LIN {X 0,Y 552.339,Z 586.998,A -85,B 0,C 180,E1 25712.762,E2 25712.762} C_VEL
LIN {X 0,Y 551.347,Z 587.125,A -85,B 0,C 180,E1 25711.964,E2 25711.964} C_VEL
LIN {X 0,Y 544.942,Z 587.913,A -85,B 0,C 180,E1 25709.72,E2 25709.72} C_VEL
LIN {X 0,Y 544.404,Z 587.984,A -85,B 0,C 180,E1 25709.136,E2 25709.136} C_VEL
LIN {X 0,Y 544.37,Z 587.986,A -85,B 0,C 180,E1 25705.803,E2 25705.803} C_VEL
LIN {X 0,Y 544.404,Z 587.987,A -85,B 0,C 180,E1 25702.428,E2 25702.428} C_VEL
LIN {X 0,Y 544.416,Z 588.083,A -85,B 0,C 180,E1 25698.94,E2 25698.94} C_VEL
LIN {X 0,Y 547.399,Z 600.07,A -85,B 0,C 180,E1 25697.246,E2 25697.246} C_VEL
LIN {X 0,Y 546.491,Z 629.146,A -85,B 0,C 180,E1 25693.756,E2 25693.756} C_VEL
LIN {X 0,Y 545.718,Z 658.309,A -85,B 0,C 180,E1 25690.342,E2 25690.342} C_VEL
LIN {X 0,Y 545.195,Z 688.021,A -85,B 0,C 180,E1 25686.98,E2 25686.98} C_VEL
LIN {X 0,Y 544.902,Z 710.009,A -85,B 0,C 180,E1 25684.567,E2 25684.567} C_VEL
LIN {X 0,Y 545.702,Z 718.325,A -85,B 0,C 180,E1 25684.417,E2 25684.417} C_VEL
LIN {X 0,Y 545.347,Z 821.497,A -85,B 0,C 180,E1 25683.028,E2 25683.028} C_VEL
LIN {X 0,Y 545.212,Z 836.514,A -85,B 0,C 180,E1 25682.627,E2 25682.627} C_VEL
LIN {X 0,Y 544.998,Z 851.155,A -85,B 0,C 180,E1 25682.019,E2 25682.019} C_VEL
LIN {X 0,Y 544.754,Z 864.801,A -85,B 0,C 180,E1 25681.232,E2 25681.232} C_VEL
LIN {X 0,Y 544.523,Z 876.818,A -85,B 0,C 180,E1 25680.329,E2 25680.329} C_VEL
LIN {X 0,Y 544.331,Z 888.046,A -85,B 0,C 180,E1 25679.248,E2 25679.248} C_VEL
LIN {X 0,Y 544.163,Z 897.795,A -85,B 0,C 180,E1 25678.059,E2 25678.059} C_VEL
LIN {X 0,Y 544.036,Z 906.382,A -85,B 0,C 180,E1 25676.721,E2 25676.721} C_VEL
LIN {X 0,Y 543.965,Z 913.553,A -85,B 0,C 180,E1 25675.242,E2 25675.242} C_VEL
LIN {X 0,Y 543.93,Z 918.751,A -85,B 0,C 180,E1 25673.732,E2 25673.732} C_VEL
LIN {X 0,Y 543.919,Z 922.084,A -85,B 0,C 180,E1 25672.252,E2 25672.252} C_VEL
LIN {X 0,Y 543.917,Z 923.807,A -85,B 0,C 180,E1 25670.662,E2 25670.662} C_VEL
LIN {X 0,Y 543.917,Z 923.713,A -85,B 0,C 180,E1 25669.099,E2 25669.099} C_VEL
LIN {X 0,Y 543.919,Z 921.897,A -85,B 0,C 180,E1 25667.546,E2 25667.546} C_VEL
LIN {X 0,Y 543.934,Z 917.94,A -85,B 0,C 180,E1 25665.896,E2 25665.896} C_VEL
LIN {X 0,Y 543.976,Z 912.247,A -85,B 0,C 180,E1 25664.367,E2 25664.367} C_VEL
LIN {X 0,Y 544.045,Z 905.689,A -85,B 0,C 180,E1 25663.065,E2 25663.065} C_VEL
LIN {X 0,Y 544.186,Z 896.405,A -85,B 0,C 180,E1 25661.66,E2 25661.66} C_VEL
LIN {X 0,Y 544.379,Z 885.783,A -85,B 0,C 180,E1 25660.423,E2 25660.423} C_VEL
LIN {X 0,Y 544.567,Z 874.019,A -85,B 0,C 180,E1 25659.351,E2 25659.351} C_VEL
LIN {X 0,Y 544.808,Z 862.012,A -85,B 0,C 180,E1 25658.496,E2 25658.496} C_VEL
LIN {X 0,Y 545.046,Z 848.15,A -85,B 0,C 180,E1 25657.749,E2 25657.749} C_VEL
LIN {X 0,Y 545.235,Z 834.039,A -85,B 0,C 180,E1 25657.204,E2 25657.204} C_VEL
LIN {X 0,Y 545.374,Z 818.941,A -85,B 0,C 180,E1 25656.832,E2 25656.832} C_VEL
LIN {X 0,Y 545.482,Z 714.402,A -85,B 0,C 180,E1 25655.434,E2 25655.434} C_VEL
LIN {X 0,Y 544.878,Z 709.572,A -85,B 0,C 180,E1 25655.317,E2 25655.317} C_VEL
LIN {X 0,Y 545.341,Z 678.781,A -85,B 0,C 180,E1 25651.891,E2 25651.891} C_VEL
LIN {X 0,Y 545.944,Z 649.394,A -85,B 0,C 180,E1 25648.531,E2 25648.531} C_VEL
LIN {X 0,Y 546.652,Z 620.644,A -85,B 0,C 180,E1 25645.173,E2 25645.173} C_VEL
LIN {X 0,Y 547.193,Z 598.729,A -85,B 0,C 180,E1 25642.545,E2 25642.545} C_VEL
LIN {X 0,Y 544.402,Z 588.081,A -85,B 0,C 180,E1 25641.018,E2 25641.018} C_VEL
LIN {X 0,Y 544.396,Z 587.986,A -85,B 0,C 180,E1 25637.591,E2 25637.591} C_VEL
LIN {X 0,Y 544.389,Z 587.981,A -85,B 0,C 180,E1 25634.117,E2 25634.117} C_VEL
LIN {X 0,Y 544.391,Z 587.983,A -85,B 0,C 180,E1 25630.743,E2 25630.743} C_VEL
LIN {X 0,Y 544.383,Z 587.984,A -85,B 0,C 180,E1 25627.426,E2 25627.426} C_VEL
LIN {X 0,Y 544.4,Z 587.979,A -85,B 0,C 180,E1 25623.962,E2 25623.962} C_VEL
LIN {X 0,Y 544.398,Z 587.974,A -85,B 0,C 180,E1 25620.513,E2 25620.513} C_VEL
LIN {X 0,Y 544.377,Z 587.976,A -85,B 0,C 180,E1 25617.191,E2 25617.191} C_VEL
LIN {X 0,Y 544.397,Z 587.98,A -85,B 0,C 180,E1 25613.874,E2 25613.874} C_VEL
LIN {X 0,Y 544.388,Z 587.986,A -85,B 0,C 180,E1 25610.48,E2 25610.48} C_VEL
LIN {X 0,Y 544.379,Z 587.976,A -85,B 0,C 180,E1 25606.971,E2 25606.971} C_VEL
LIN {X 0,Y 544.399,Z 587.983,A -85,B 0,C 180,E1 25603.644,E2 25603.644} C_VEL
LIN {X 0,Y 544.372,Z 587.978,A -85,B 0,C 180,E1 25600.281,E2 25600.281} C_VEL
LIN {X 0,Y 544.399,Z 587.979,A -85,B 0,C 180,E1 25596.912,E2 25596.912} C_VEL
LIN {X 0,Y 544.405,Z 587.979,A -85,B 0,C 180,E1 25593.435,E2 25593.435} C_VEL
LIN {X 0,Y 544.368,Z 587.984,A -85,B 0,C 180,E1 25590.095,E2 25590.095} C_VEL
LIN {X 0,Y 544.401,Z 587.972,A -85,B 0,C 180,E1 25586.797,E2 25586.797} C_VEL
LIN {X 0,Y 544.37,Z 587.983,A -85,B 0,C 180,E1 25583.489,E2 25583.489} C_VEL
LIN {X 0,Y 544.387,Z 587.978,A -85,B 0,C 180,E1 25580.088,E2 25580.088} C_VEL
LIN {X 0,Y 544.402,Z 587.979,A -85,B 0,C 180,E1 25576.759,E2 25576.759} C_VEL
LIN {X 0,Y 544.364,Z 587.983,A -85,B 0,C 180,E1 25573.49,E2 25573.49} C_VEL
LIN {X 0,Y 544.402,Z 587.973,A -85,B 0,C 180,E1 25570.155,E2 25570.155} C_VEL
LIN {X 0,Y 544.361,Z 587.982,A -85,B 0,C 180,E1 25566.857,E2 25566.857} C_VEL
LIN {X 0,Y 544.387,Z 587.979,A -85,B 0,C 180,E1 25563.475,E2 25563.475} C_VEL
LIN {X 0,Y 544.404,Z 587.978,A -85,B 0,C 180,E1 25560.105,E2 25560.105} C_VEL
LIN {X 0,Y 544.358,Z 587.984,A -85,B 0,C 180,E1 25556.841,E2 25556.841} C_VEL
LIN {X 0,Y 544.406,Z 587.973,A -85,B 0,C 180,E1 25553.521,E2 25553.521} C_VEL
LIN {X 0,Y 544.353,Z 587.985,A -85,B 0,C 180,E1 25550.271,E2 25550.271} C_VEL
LIN {X 0,Y 544.395,Z 587.977,A -85,B 0,C 180,E1 25546.944,E2 25546.944} C_VEL
LIN {X 0,Y 544.373,Z 587.985,A -85,B 0,C 180,E1 25543.679,E2 25543.679} C_VEL
LIN {X 0,Y 544.359,Z 587.981,A -85,B 0,C 180,E1 25540.247,E2 25540.247} C_VEL
LIN {X 0,Y 544.409,Z 587.984,A -85,B 0,C 180,E1 25536.947,E2 25536.947} C_VEL
LIN {X 0,Y 544.346,Z 587.982,A -85,B 0,C 180,E1 25533.685,E2 25533.685} C_VEL
LIN {X 0,Y 544.406,Z 587.979,A -85,B 0,C 180,E1 25530.393,E2 25530.393} C_VEL
LIN {X 0,Y 544.355,Z 587.988,A -85,B 0,C 180,E1 25527.191,E2 25527.191} C_VEL
LIN {X 0,Y 544.362,Z 587.984,A -85,B 0,C 180,E1 25523.74,E2 25523.74} C_VEL
LIN {X 0,Y 544.405,Z 587.986,A -85,B 0,C 180,E1 25520.478,E2 25520.478} C_VEL
LIN {X 0,Y 544.342,Z 587.987,A -85,B 0,C 180,E1 25517.186,E2 25517.186} C_VEL
LIN {X 0,Y 544.409,Z 587.983,A -85,B 0,C 180,E1 25513.95,E2 25513.95} C_VEL
LIN {X 0,Y 544.343,Z 587.988,A -85,B 0,C 180,E1 25510.698,E2 25510.698} C_VEL
LIN {X 0,Y 544.397,Z 587.982,A -85,B 0,C 180,E1 25507.44,E2 25507.44} C_VEL
LIN {X 0,Y 544.362,Z 587.993,A -85,B 0,C 180,E1 25504.198,E2 25504.198} C_VEL
LIN {X 0,Y 544.39,Z 588.207,A -85,B 0,C 180,E1 25502.928,E2 25502.928} C_VEL
LIN {X 0,Y 549.723,Z 603.754,A -85,B 0,C 180,E1 25501.345,E2 25501.345} C_VEL
LIN {X 0,Y 548.818,Z 646.737,A -85,B 0,C 180,E1 25498.214,E2 25498.214} C_VEL
LIN {X 0,Y 547.856,Z 691.846,A -85,B 0,C 180,E1 25494.939,E2 25494.939} C_VEL
LIN {X 0,Y 549.107,Z 701.947,A -85,B 0,C 180,E1 25494.729,E2 25494.729} C_VEL
LIN {X 0,Y 548.003,Z 901.303,A -85,B 0,C 180,E1 25491.965,E2 25491.965} C_VEL
LIN {X 0,Y 547.684,Z 920.34,A -85,B 0,C 180,E1 25491.503,E2 25491.503} C_VEL
LIN {X 0,Y 547.305,Z 938.39,A -85,B 0,C 180,E1 25490.87,E2 25490.87} C_VEL
LIN {X 0,Y 546.826,Z 956.036,A -85,B 0,C 180,E1 25490.05,E2 25490.05} C_VEL
LIN {X 0,Y 546.332,Z 972.766,A -85,B 0,C 180,E1 25489.068,E2 25489.068} C_VEL
LIN {X 0,Y 545.854,Z 988.622,A -85,B 0,C 180,E1 25487.923,E2 25487.923} C_VEL
LIN {X 0,Y 545.378,Z 1003.553,A -85,B 0,C 180,E1 25486.619,E2 25486.619} C_VEL
LIN {X 0,Y 544.956,Z 1017.225,A -85,B 0,C 180,E1 25485.186,E2 25485.186} C_VEL
LIN {X 0,Y 544.601,Z 1029.912,A -85,B 0,C 180,E1 25483.592,E2 25483.592} C_VEL
LIN {X 0,Y 544.329,Z 1041.229,A -85,B 0,C 180,E1 25481.872,E2 25481.872} C_VEL
LIN {X 0,Y 544.129,Z 1050.993,A -85,B 0,C 180,E1 25480.054,E2 25480.054} C_VEL
LIN {X 0,Y 544.004,Z 1059.176,A -85,B 0,C 180,E1 25478.136,E2 25478.136} C_VEL
LIN {X 0,Y 543.949,Z 1065.412,A -85,B 0,C 180,E1 25476.226,E2 25476.226} C_VEL
LIN {X 0,Y 543.923,Z 1069.877,A -85,B 0,C 180,E1 25474.323,E2 25474.323} C_VEL
LIN {X 0,Y 543.914,Z 1072.792,A -85,B 0,C 180,E1 25472.318,E2 25472.318} C_VEL
LIN {X 0,Y 543.908,Z 1073.94,A -85,B 0,C 180,E1 25470.316,E2 25470.316} C_VEL
LIN {X 0,Y 543.913,Z 1073.347,A -85,B 0,C 180,E1 25468.315,E2 25468.315} C_VEL
LIN {X 0,Y 543.915,Z 1071.003,A -85,B 0,C 180,E1 25466.311,E2 25466.311} C_VEL
LIN {X 0,Y 543.931,Z 1067.098,A -85,B 0,C 180,E1 25464.409,E2 25464.409} C_VEL
LIN {X 0,Y 543.981,Z 1061.468,A -85,B 0,C 180,E1 25462.502,E2 25462.502} C_VEL
LIN {X 0,Y 544.074,Z 1054.427,A -85,B 0,C 180,E1 25460.693,E2 25460.693} C_VEL
LIN {X 0,Y 544.236,Z 1045.516,A -85,B 0,C 180,E1 25458.878,E2 25458.878} C_VEL
LIN {X 0,Y 544.47,Z 1035.153,A -85,B 0,C 180,E1 25457.162,E2 25457.162} C_VEL
LIN {X 0,Y 544.779,Z 1023.351,A -85,B 0,C 180,E1 25455.546,E2 25455.546} C_VEL
LIN {X 0,Y 545.178,Z 1010.082,A -85,B 0,C 180,E1 25454.032,E2 25454.032} C_VEL
LIN {X 0,Y 545.649,Z 995.223,A -85,B 0,C 180,E1 25452.621,E2 25452.621} C_VEL
LIN {X 0,Y 546.157,Z 979.233,A -85,B 0,C 180,E1 25451.37,E2 25451.37} C_VEL
LIN {X 0,Y 546.64,Z 962.05,A -85,B 0,C 180,E1 25450.277,E2 25450.277} C_VEL
LIN {X 0,Y 547.142,Z 944.807,A -85,B 0,C 180,E1 25449.404,E2 25449.404} C_VEL
LIN {X 0,Y 547.55,Z 926.53,A -85,B 0,C 180,E1 25448.692,E2 25448.692} C_VEL
LIN {X 0,Y 547.897,Z 907.921,A -85,B 0,C 180,E1 25448.174,E2 25448.174} C_VEL
LIN {X 0,Y 548.116,Z 887.491,A -85,B 0,C 180,E1 25447.82,E2 25447.82} C_VEL
LIN {X 0,Y 548.951,Z 699.141,A -85,B 0,C 180,E1 25445.224,E2 25445.224} C_VEL
LIN {X 0,Y 547.831,Z 691.329,A -85,B 0,C 180,E1 25445.035,E2 25445.035} C_VEL
LIN {X 0,Y 548.818,Z 646.743,A -85,B 0,C 180,E1 25441.786,E2 25441.786} C_VEL
LIN {X 0,Y 549.723,Z 603.759,A -85,B 0,C 180,E1 25438.655,E2 25438.655} C_VEL
LIN {X 0,Y 544.405,Z 588.322,A -85,B 0,C 180,E1 25437.1,E2 25437.1} C_VEL
LIN {X 0,Y 544.403,Z 587.985,A -85,B 0,C 180,E1 25436.303,E2 25436.303} C_VEL
LIN {X 0,Y 544.347,Z 587.99,A -85,B 0,C 180,E1 25433.085,E2 25433.085} C_VEL
LIN {X 0,Y 544.374,Z 587.989,A -85,B 0,C 180,E1 25429.72,E2 25429.72} C_VEL
LIN {X 0,Y 544.375,Z 587.983,A -85,B 0,C 180,E1 25426.51,E2 25426.51} C_VEL
LIN {X 0,Y 544.348,Z 587.99,A -85,B 0,C 180,E1 25423.18,E2 25423.18} C_VEL
LIN {X 0,Y 544.408,Z 587.982,A -85,B 0,C 180,E1 25420.002,E2 25420.002} C_VEL
LIN {X 0,Y 544.342,Z 587.988,A -85,B 0,C 180,E1 25416.784,E2 25416.784} C_VEL
LIN {X 0,Y 544.407,Z 587.984,A -85,B 0,C 180,E1 25413.56,E2 25413.56} C_VEL
LIN {X 0,Y 544.348,Z 587.986,A -85,B 0,C 180,E1 25410.311,E2 25410.311} C_VEL
LIN {X 0,Y 544.39,Z 587.986,A -85,B 0,C 180,E1 25406.978,E2 25406.978} C_VEL
LIN {X 0,Y 544.369,Z 587.98,A -85,B 0,C 180,E1 25403.718,E2 25403.718} C_VEL
LIN {X 0,Y 544.352,Z 587.985,A -85,B 0,C 180,E1 25400.313,E2 25400.313} C_VEL
LIN {X 0,Y 544.405,Z 587.981,A -85,B 0,C 180,E1 25397.089,E2 25397.089} C_VEL
LIN {X 0,Y 544.349,Z 587.983,A -85,B 0,C 180,E1 25393.815,E2 25393.815} C_VEL
LIN {X 0,Y 544.406,Z 587.986,A -85,B 0,C 180,E1 25390.583,E2 25390.583} C_VEL
LIN {X 0,Y 544.359,Z 587.984,A -85,B 0,C 180,E1 25387.281,E2 25387.281} C_VEL
LIN {X 0,Y 544.366,Z 587.987,A -85,B 0,C 180,E1 25383.791,E2 25383.791} C_VEL
LIN {X 0,Y 544.402,Z 587.98,A -85,B 0,C 180,E1 25380.526,E2 25380.526} C_VEL
LIN {X 0,Y 544.357,Z 587.985,A -85,B 0,C 180,E1 25377.157,E2 25377.157} C_VEL
LIN {X 0,Y 544.405,Z 587.984,A -85,B 0,C 180,E1 25373.779,E2 25373.779} C_VEL
LIN {X 0,Y 544.371,Z 587.977,A -85,B 0,C 180,E1 25370.485,E2 25370.485} C_VEL
LIN {X 0,Y 544.37,Z 587.982,A -85,B 0,C 180,E1 25367.051,E2 25367.051} C_VEL
LIN {X 0,Y 544.405,Z 587.982,A -85,B 0,C 180,E1 25363.789,E2 25363.789} C_VEL
LIN {X 0,Y 544.364,Z 587.984,A -85,B 0,C 180,E1 25360.434,E2 25360.434} C_VEL
LIN {X 0,Y 544.404,Z 587.987,A -85,B 0,C 180,E1 25357.085,E2 25357.085} C_VEL
LIN {X 0,Y 544.387,Z 587.982,A -85,B 0,C 180,E1 25353.675,E2 25353.675} C_VEL
LIN {X 0,Y 544.374,Z 587.986,A -85,B 0,C 180,E1 25350.27,E2 25350.27} C_VEL
LIN {X 0,Y 544.404,Z 587.984,A -85,B 0,C 180,E1 25349.136,E2 25349.136} C_VEL
LIN {X 0,Y 543.395,Z 588.116,A -85,B 0,C 180,E1 25348.325,E2 25348.325} C_VEL
LIN {X 0,Y 536.947,Z 588.912,A -85,B 0,C 180,E1 25346.048,E2 25346.048} C_VEL
LIN {X 0,Y 536.441,Z 588.974,A -85,B 0,C 180,E1 25345.455,E2 25345.455} C_VEL
LIN {X 0,Y 536.444,Z 588.977,A -85,B 0,C 180,E1 25342.038,E2 25342.038} C_VEL
LIN {X 0,Y 536.48,Z 589.253,A -85,B 0,C 180,E1 25339.273,E2 25339.273} C_VEL
LIN {X 0,Y 539.882,Z 602.566,A -85,B 0,C 180,E1 25337.39,E2 25337.39} C_VEL
LIN {X 0,Y 538.894,Z 630.944,A -85,B 0,C 180,E1 25333.941,E2 25333.941} C_VEL
LIN {X 0,Y 538.069,Z 659.803,A -85,B 0,C 180,E1 25330.534,E2 25330.534} C_VEL
LIN {X 0,Y 537.369,Z 688.964,A -85,B 0,C 180,E1 25327.128,E2 25327.128} C_VEL
LIN {X 0,Y 537.043,Z 710,A -85,B 0,C 180,E1 25324.786,E2 25324.786} C_VEL
LIN {X 0,Y 537.954,Z 718.938,A -85,B 0,C 180,E1 25324.622,E2 25324.622} C_VEL
LIN {X 0,Y 537.554,Z 821.421,A -85,B 0,C 180,E1 25323.222,E2 25323.222} C_VEL
LIN {X 0,Y 537.403,Z 836.215,A -85,B 0,C 180,E1 25322.825,E2 25322.825} C_VEL
LIN {X 0,Y 537.158,Z 851.048,A -85,B 0,C 180,E1 25322.203,E2 25322.203} C_VEL
LIN {X 0,Y 536.887,Z 864.354,A -85,B 0,C 180,E1 25321.43,E2 25321.43} C_VEL
LIN {X 0,Y 536.626,Z 876.448,A -85,B 0,C 180,E1 25320.516,E2 25320.516} C_VEL
LIN {X 0,Y 536.391,Z 888.326,A -85,B 0,C 180,E1 25319.357,E2 25319.357} C_VEL
LIN {X 0,Y 536.194,Z 898.279,A -85,B 0,C 180,E1 25318.112,E2 25318.112} C_VEL
LIN {X 0,Y 536.057,Z 906.33,A -85,B 0,C 180,E1 25316.832,E2 25316.832} C_VEL
LIN {X 0,Y 535.972,Z 913.681,A -85,B 0,C 180,E1 25315.29,E2 25315.29} C_VEL
LIN {X 0,Y 535.931,Z 918.819,A -85,B 0,C 180,E1 25313.765,E2 25313.765} C_VEL
LIN {X 0,Y 535.919,Z 922.13,A -85,B 0,C 180,E1 25312.255,E2 25312.255} C_VEL
LIN {X 0,Y 535.917,Z 923.823,A -85,B 0,C 180,E1 25310.647,E2 25310.647} C_VEL
LIN {X 0,Y 535.917,Z 923.693,A -85,B 0,C 180,E1 25309.056,E2 25309.056} C_VEL
LIN {X 0,Y 535.919,Z 921.841,A -85,B 0,C 180,E1 25307.48,E2 25307.48} C_VEL
LIN {X 0,Y 535.937,Z 917.856,A -85,B 0,C 180,E1 25305.806,E2 25305.806} C_VEL
LIN {X 0,Y 535.987,Z 912.124,A -85,B 0,C 180,E1 25304.255,E2 25304.255} C_VEL
LIN {X 0,Y 536.079,Z 904.873,A -85,B 0,C 180,E1 25302.824,E2 25302.824} C_VEL
LIN {X 0,Y 536.235,Z 896.202,A -85,B 0,C 180,E1 25301.508,E2 25301.508} C_VEL
LIN {X 0,Y 536.459,Z 885.314,A -85,B 0,C 180,E1 25300.231,E2 25300.231} C_VEL
LIN {X 0,Y 536.674,Z 873.672,A -85,B 0,C 180,E1 25299.166,E2 25299.166} C_VEL
LIN {X 0,Y 536.953,Z 861.56,A -85,B 0,C 180,E1 25298.297,E2 25298.297} C_VEL
LIN {X 0,Y 537.22,Z 847.556,A -85,B 0,C 180,E1 25297.54,E2 25297.54} C_VEL
LIN {X 0,Y 537.437,Z 833.184,A -85,B 0,C 180,E1 25296.989,E2 25296.989} C_VEL
LIN {X 0,Y 537.584,Z 818.438,A -85,B 0,C 180,E1 25296.631,E2 25296.631} C_VEL
LIN {X 0,Y 537.734,Z 715.162,A -85,B 0,C 180,E1 25295.231,E2 25295.231} C_VEL
LIN {X 0,Y 537.018,Z 709.61,A -85,B 0,C 180,E1 25295.1,E2 25295.1} C_VEL
LIN {X 0,Y 537.551,Z 679.59,A -85,B 0,C 180,E1 25291.705,E2 25291.705} C_VEL
LIN {X 0,Y 538.301,Z 650.522,A -85,B 0,C 180,E1 25288.297,E2 25288.297} C_VEL
LIN {X 0,Y 539.049,Z 622.508,A -85,B 0,C 180,E1 25284.998,E2 25284.998} C_VEL
LIN {X 0,Y 539.663,Z 601.17,A -85,B 0,C 180,E1 25282.405,E2 25282.405} C_VEL
LIN {X 0,Y 536.476,Z 589.085,A -85,B 0,C 180,E1 25280.649,E2 25280.649} C_VEL
LIN {X 0,Y 536.456,Z 588.977,A -85,B 0,C 180,E1 25277.185,E2 25277.185} C_VEL
LIN {X 0,Y 536.443,Z 588.972,A -85,B 0,C 180,E1 25273.876,E2 25273.876} C_VEL
LIN {X 0,Y 536.455,Z 588.969,A -85,B 0,C 180,E1 25270.511,E2 25270.511} C_VEL
LIN {X 0,Y 536.459,Z 588.965,A -85,B 0,C 180,E1 25267.074,E2 25267.074} C_VEL
LIN {X 0,Y 536.447,Z 588.969,A -85,B 0,C 180,E1 25263.666,E2 25263.666} C_VEL
LIN {X 0,Y 536.455,Z 588.958,A -85,B 0,C 180,E1 25260.278,E2 25260.278} C_VEL
LIN {X 0,Y 536.443,Z 588.966,A -85,B 0,C 180,E1 25256.899,E2 25256.899} C_VEL
LIN {X 0,Y 536.454,Z 588.967,A -85,B 0,C 180,E1 25253.448,E2 25253.448} C_VEL
LIN {X 0,Y 536.464,Z 588.976,A -85,B 0,C 180,E1 25250.122,E2 25250.122} C_VEL
LIN {X 0,Y 536.435,Z 588.966,A -85,B 0,C 180,E1 25246.692,E2 25246.692} C_VEL
LIN {X 0,Y 536.462,Z 588.968,A -85,B 0,C 180,E1 25243.305,E2 25243.305} C_VEL
LIN {X 0,Y 536.462,Z 588.969,A -85,B 0,C 180,E1 25239.835,E2 25239.835} C_VEL
LIN {X 0,Y 536.436,Z 588.971,A -85,B 0,C 180,E1 25236.483,E2 25236.483} C_VEL
LIN {X 0,Y 536.462,Z 588.966,A -85,B 0,C 180,E1 25233.1,E2 25233.1} C_VEL
LIN {X 0,Y 536.434,Z 588.976,A -85,B 0,C 180,E1 25229.723,E2 25229.723} C_VEL
LIN {X 0,Y 536.439,Z 588.96,A -85,B 0,C 180,E1 25226.215,E2 25226.215} C_VEL
LIN {X 0,Y 536.464,Z 588.973,A -85,B 0,C 180,E1 25222.81,E2 25222.81} C_VEL
LIN {X 0,Y 536.426,Z 588.972,A -85,B 0,C 180,E1 25219.49,E2 25219.49} C_VEL
LIN {X 0,Y 536.462,Z 588.964,A -85,B 0,C 180,E1 25216.124,E2 25216.124} C_VEL
LIN {X 0,Y 536.457,Z 588.978,A -85,B 0,C 180,E1 25212.705,E2 25212.705} C_VEL
LIN {X 0,Y 536.423,Z 588.963,A -85,B 0,C 180,E1 25209.333,E2 25209.333} C_VEL
LIN {X 0,Y 536.465,Z 588.97,A -85,B 0,C 180,E1 25205.991,E2 25205.991} C_VEL
LIN {X 0,Y 536.423,Z 588.974,A -85,B 0,C 180,E1 25202.671,E2 25202.671} C_VEL
LIN {X 0,Y 536.441,Z 588.965,A -85,B 0,C 180,E1 25199.253,E2 25199.253} C_VEL
LIN {X 0,Y 536.463,Z 588.976,A -85,B 0,C 180,E1 25195.939,E2 25195.939} C_VEL
LIN {X 0,Y 536.414,Z 588.964,A -85,B 0,C 180,E1 25192.586,E2 25192.586} C_VEL
LIN {X 0,Y 536.466,Z 588.971,A -85,B 0,C 180,E1 25189.259,E2 25189.259} C_VEL
LIN {X 0,Y 536.416,Z 588.973,A -85,B 0,C 180,E1 25185.977,E2 25185.977} C_VEL
LIN {X 0,Y 536.433,Z 588.972,A -85,B 0,C 180,E1 25182.537,E2 25182.537} C_VEL
LIN {X 0,Y 536.461,Z 588.97,A -85,B 0,C 180,E1 25179.26,E2 25179.26} C_VEL
LIN {X 0,Y 536.411,Z 588.974,A -85,B 0,C 180,E1 25175.974,E2 25175.974} C_VEL
LIN {X 0,Y 536.471,Z 588.972,A -85,B 0,C 180,E1 25172.711,E2 25172.711} C_VEL
LIN {X 0,Y 536.407,Z 588.975,A -85,B 0,C 180,E1 25169.449,E2 25169.449} C_VEL
LIN {X 0,Y 536.455,Z 588.969,A -85,B 0,C 180,E1 25166.132,E2 25166.132} C_VEL
LIN {X 0,Y 536.432,Z 588.979,A -85,B 0,C 180,E1 25162.85,E2 25162.85} C_VEL
LIN {X 0,Y 536.417,Z 588.975,A -85,B 0,C 180,E1 25159.509,E2 25159.509} C_VEL
LIN {X 0,Y 536.465,Z 588.974,A -85,B 0,C 180,E1 25156.254,E2 25156.254} C_VEL
LIN {X 0,Y 536.404,Z 588.975,A -85,B 0,C 180,E1 25153.018,E2 25153.018} C_VEL
LIN {X 0,Y 536.471,Z 588.973,A -85,B 0,C 180,E1 25149.738,E2 25149.738} C_VEL
LIN {X 0,Y 536.409,Z 588.977,A -85,B 0,C 180,E1 25146.485,E2 25146.485} C_VEL
LIN {X 0,Y 536.494,Z 589.204,A -85,B 0,C 180,E1 25143.353,E2 25143.353} C_VEL
LIN {X 0,Y 542.364,Z 606.653,A -85,B 0,C 180,E1 25141.541,E2 25141.541} C_VEL
LIN {X 0,Y 541.321,Z 650.057,A -85,B 0,C 180,E1 25138.34,E2 25138.34} C_VEL
LIN {X 0,Y 540.456,Z 692.127,A -85,B 0,C 180,E1 25135.298,E2 25135.298} C_VEL
LIN {X 0,Y 541.836,Z 702.965,A -85,B 0,C 180,E1 25135.069,E2 25135.069} C_VEL
LIN {X 0,Y 540.577,Z 901.465,A -85,B 0,C 180,E1 25132.279,E2 25132.279} C_VEL
LIN {X 0,Y 540.22,Z 920.446,A -85,B 0,C 180,E1 25131.812,E2 25131.812} C_VEL
LIN {X 0,Y 539.79,Z 938.389,A -85,B 0,C 180,E1 25131.174,E2 25131.174} C_VEL
LIN {X 0,Y 539.254,Z 956.034,A -85,B 0,C 180,E1 25130.344,E2 25130.344} C_VEL
LIN {X 0,Y 538.689,Z 972.764,A -85,B 0,C 180,E1 25129.349,E2 25129.349} C_VEL
LIN {X 0,Y 538.124,Z 989.196,A -85,B 0,C 180,E1 25128.141,E2 25128.141} C_VEL
LIN {X 0,Y 537.583,Z 1004.107,A -85,B 0,C 180,E1 25126.811,E2 25126.811} C_VEL
LIN {X 0,Y 537.094,Z 1017.942,A -85,B 0,C 180,E1 25125.329,E2 25125.329} C_VEL
LIN {X 0,Y 536.688,Z 1030.682,A -85,B 0,C 180,E1 25123.686,E2 25123.686} C_VEL
LIN {X 0,Y 536.38,Z 1041.863,A -85,B 0,C 180,E1 25121.942,E2 25121.942} C_VEL
LIN {X 0,Y 536.155,Z 1051.507,A -85,B 0,C 180,E1 25120.096,E2 25120.096} C_VEL
LIN {X 0,Y 536.023,Z 1059.176,A -85,B 0,C 180,E1 25118.258,E2 25118.258} C_VEL
LIN {X 0,Y 535.955,Z 1065.412,A -85,B 0,C 180,E1 25116.319,E2 25116.319} C_VEL
LIN {X 0,Y 535.924,Z 1069.878,A -85,B 0,C 180,E1 25114.387,E2 25114.387} C_VEL
LIN {X 0,Y 535.913,Z 1072.793,A -85,B 0,C 180,E1 25112.353,E2 25112.353} C_VEL
LIN {X 0,Y 535.908,Z 1073.94,A -85,B 0,C 180,E1 25110.321,E2 25110.321} C_VEL
LIN {X 0,Y 535.912,Z 1073.347,A -85,B 0,C 180,E1 25108.29,E2 25108.29} C_VEL
LIN {X 0,Y 535.916,Z 1071.002,A -85,B 0,C 180,E1 25106.256,E2 25106.256} C_VEL
LIN {X 0,Y 535.935,Z 1067.097,A -85,B 0,C 180,E1 25104.326,E2 25104.326} C_VEL
LIN {X 0,Y 535.995,Z 1061.468,A -85,B 0,C 180,E1 25102.389,E2 25102.389} C_VEL
LIN {X 0,Y 536.098,Z 1054.427,A -85,B 0,C 180,E1 25100.554,E2 25100.554} C_VEL
LIN {X 0,Y 536.288,Z 1045.517,A -85,B 0,C 180,E1 25098.711,E2 25098.711} C_VEL
LIN {X 0,Y 536.559,Z 1035.154,A -85,B 0,C 180,E1 25096.969,E2 25096.969} C_VEL
LIN {X 0,Y 536.916,Z 1023.352,A -85,B 0,C 180,E1 25095.329,E2 25095.329} C_VEL
LIN {X 0,Y 537.394,Z 1009.682,A -85,B 0,C 180,E1 25093.751,E2 25093.751} C_VEL
LIN {X 0,Y 537.944,Z 994.604,A -85,B 0,C 180,E1 25092.309,E2 25092.309} C_VEL
LIN {X 0,Y 538.519,Z 978.437,A -85,B 0,C 180,E1 25091.039,E2 25091.039} C_VEL
LIN {X 0,Y 539.059,Z 961.783,A -85,B 0,C 180,E1 25089.973,E2 25089.973} C_VEL
LIN {X 0,Y 539.611,Z 944.808,A -85,B 0,C 180,E1 25089.103,E2 25089.103} C_VEL
LIN {X 0,Y 540.071,Z 926.533,A -85,B 0,C 180,E1 25088.382,E2 25088.382} C_VEL
LIN {X 0,Y 540.462,Z 907.852,A -85,B 0,C 180,E1 25087.857,E2 25087.857} C_VEL
LIN {X 0,Y 540.711,Z 887.237,A -85,B 0,C 180,E1 25087.496,E2 25087.496} C_VEL
LIN {X 0,Y 541.681,Z 700.18,A -85,B 0,C 180,E1 25084.883,E2 25084.883} C_VEL
LIN {X 0,Y 540.398,Z 691.33,A -85,B 0,C 180,E1 25084.668,E2 25084.668} C_VEL
LIN {X 0,Y 541.366,Z 647.713,A -85,B 0,C 180,E1 25081.488,E2 25081.488} C_VEL
LIN {X 0,Y 542.369,Z 606.454,A -85,B 0,C 180,E1 25078.444,E2 25078.444} C_VEL
LIN {X 0,Y 536.504,Z 589.279,A -85,B 0,C 180,E1 25076.669,E2 25076.669} C_VEL
LIN {X 0,Y 536.404,Z 588.98,A -85,B 0,C 180,E1 25075.476,E2 25075.476} C_VEL
LIN {X 0,Y 536.47,Z 588.973,A -85,B 0,C 180,E1 25072.18,E2 25072.18} C_VEL
LIN {X 0,Y 536.403,Z 588.976,A -85,B 0,C 180,E1 25068.995,E2 25068.995} C_VEL
LIN {X 0,Y 536.444,Z 588.98,A -85,B 0,C 180,E1 25065.657,E2 25065.657} C_VEL
LIN {X 0,Y 536.43,Z 588.974,A -85,B 0,C 180,E1 25062.429,E2 25062.429} C_VEL
LIN {X 0,Y 536.41,Z 588.974,A -85,B 0,C 180,E1 25059.052,E2 25059.052} C_VEL
LIN {X 0,Y 536.465,Z 588.972,A -85,B 0,C 180,E1 25055.819,E2 25055.819} C_VEL
LIN {X 0,Y 536.405,Z 588.975,A -85,B 0,C 180,E1 25052.592,E2 25052.592} C_VEL
LIN {X 0,Y 536.47,Z 588.974,A -85,B 0,C 180,E1 25049.352,E2 25049.352} C_VEL
LIN {X 0,Y 536.414,Z 588.974,A -85,B 0,C 180,E1 25046.047,E2 25046.047} C_VEL
LIN {X 0,Y 536.436,Z 588.977,A -85,B 0,C 180,E1 25042.687,E2 25042.687} C_VEL
LIN {X 0,Y 536.444,Z 588.968,A -85,B 0,C 180,E1 25039.418,E2 25039.418} C_VEL
LIN {X 0,Y 536.414,Z 588.975,A -85,B 0,C 180,E1 25036.125,E2 25036.125} C_VEL
LIN {X 0,Y 536.465,Z 588.968,A -85,B 0,C 180,E1 25032.899,E2 25032.899} C_VEL
LIN {X 0,Y 536.414,Z 588.967,A -85,B 0,C 180,E1 25029.549,E2 25029.549} C_VEL
LIN {X 0,Y 536.456,Z 588.975,A -85,B 0,C 180,E1 25026.206,E2 25026.206} C_VEL
LIN {X 0,Y 536.436,Z 588.971,A -85,B 0,C 180,E1 25022.884,E2 25022.884} C_VEL
LIN {X 0,Y 536.422,Z 588.973,A -85,B 0,C 180,E1 25019.466,E2 25019.466} C_VEL
LIN {X 0,Y 536.465,Z 588.973,A -85,B 0,C 180,E1 25016.153,E2 25016.153} C_VEL
LIN {X 0,Y 536.421,Z 588.974,A -85,B 0,C 180,E1 25012.826,E2 25012.826} C_VEL
LIN {X 0,Y 536.457,Z 588.976,A -85,B 0,C 180,E1 25009.475,E2 25009.475} C_VEL
LIN {X 0,Y 536.452,Z 588.965,A -85,B 0,C 180,E1 25006.088,E2 25006.088} C_VEL
LIN {X 0,Y 536.428,Z 588.972,A -85,B 0,C 180,E1 25002.76,E2 25002.76} C_VEL
LIN {X 0,Y 536.464,Z 588.973,A -85,B 0,C 180,E1 24999.488,E2 24999.488} C_VEL
LIN {X 0,Y 536.426,Z 588.969,A -85,B 0,C 180,E1 24996.142,E2 24996.142} C_VEL
LIN {X 0,Y 536.458,Z 588.975,A -85,B 0,C 180,E1 24992.709,E2 24992.709} C_VEL
LIN {X 0,Y 536.465,Z 588.972,A -85,B 0,C 180,E1 24989.291,E2 24989.291} C_VEL
LIN {X 0,Y 536.431,Z 588.975,A -85,B 0,C 180,E1 24985.872,E2 24985.872} C_VEL
LIN {X 0,Y 536.441,Z 588.974,A -85,B 0,C 180,E1 24985.455,E2 24985.455} C_VEL
LIN {X 0,Y 535.483,Z 589.097,A -85,B 0,C 180,E1 24984.632,E2 24984.632} C_VEL
LIN {X 0,Y 528.936,Z 589.915,A -85,B 0,C 180,E1 24982.261,E2 24982.261} C_VEL
LIN {X 0,Y 528.494,Z 589.966,A -85,B 0,C 180,E1 24981.718,E2 24981.718} C_VEL
LIN {X 0,Y 528.538,Z 590.254,A -85,B 0,C 180,E1 24979.679,E2 24979.679} C_VEL
LIN {X 0,Y 532.378,Z 604.805,A -85,B 0,C 180,E1 24977.569,E2 24977.569} C_VEL
LIN {X 0,Y 531.299,Z 633.626,A -85,B 0,C 180,E1 24974.036,E2 24974.036} C_VEL
LIN {X 0,Y 530.389,Z 662.312,A -85,B 0,C 180,E1 24970.61,E2 24970.61} C_VEL
LIN {X 0,Y 529.589,Z 691.276,A -85,B 0,C 180,E1 24967.168,E2 24967.168} C_VEL
LIN {X 0,Y 529.194,Z 709.719,A -85,B 0,C 180,E1 24965.04,E2 24965.04} C_VEL
LIN {X 0,Y 530.216,Z 719.507,A -85,B 0,C 180,E1 24964.834,E2 24964.834} C_VEL
LIN {X 0,Y 529.766,Z 821.526,A -85,B 0,C 180,E1 24963.419,E2 24963.419} C_VEL
LIN {X 0,Y 529.59,Z 836.477,A -85,B 0,C 180,E1 24963.008,E2 24963.008} C_VEL
LIN {X 0,Y 529.311,Z 851.672,A -85,B 0,C 180,E1 24962.357,E2 24962.357} C_VEL
LIN {X 0,Y 528.993,Z 865.561,A -85,B 0,C 180,E1 24961.521,E2 24961.521} C_VEL
LIN {X 0,Y 528.697,Z 877.518,A -85,B 0,C 180,E1 24960.579,E2 24960.579} C_VEL
LIN {X 0,Y 528.444,Z 888.976,A -85,B 0,C 180,E1 24959.427,E2 24959.427} C_VEL
LIN {X 0,Y 528.217,Z 899.21,A -85,B 0,C 180,E1 24958.104,E2 24958.104} C_VEL
LIN {X 0,Y 528.065,Z 907.13,A -85,B 0,C 180,E1 24956.785,E2 24956.785} C_VEL
LIN {X 0,Y 527.979,Z 913.804,A -85,B 0,C 180,E1 24955.34,E2 24955.34} C_VEL
LIN {X 0,Y 527.932,Z 919.235,A -85,B 0,C 180,E1 24953.673,E2 24953.673} C_VEL
LIN {X 0,Y 527.921,Z 922.348,A -85,B 0,C 180,E1 24952.142,E2 24952.142} C_VEL
LIN {X 0,Y 527.917,Z 923.891,A -85,B 0,C 180,E1 24950.511,E2 24950.511} C_VEL
LIN {X 0,Y 527.918,Z 923.53,A -85,B 0,C 180,E1 24948.782,E2 24948.782} C_VEL
LIN {X 0,Y 527.92,Z 921.353,A -85,B 0,C 180,E1 24947.185,E2 24947.185} C_VEL
LIN {X 0,Y 527.944,Z 917.412,A -85,B 0,C 180,E1 24945.6,E2 24945.6} C_VEL
LIN {X 0,Y 528.006,Z 911.53,A -85,B 0,C 180,E1 24944.027,E2 24944.027} C_VEL
LIN {X 0,Y 528.117,Z 904.058,A -85,B 0,C 180,E1 24942.575,E2 24942.575} C_VEL
LIN {X 0,Y 528.305,Z 895.138,A -85,B 0,C 180,E1 24941.241,E2 24941.241} C_VEL
LIN {X 0,Y 528.558,Z 884.207,A -85,B 0,C 180,E1 24939.967,E2 24939.967} C_VEL
LIN {X 0,Y 528.822,Z 871.979,A -85,B 0,C 180,E1 24938.864,E2 24938.864} C_VEL
LIN {X 0,Y 529.142,Z 859.292,A -85,B 0,C 180,E1 24937.983,E2 24937.983} C_VEL
LIN {X 0,Y 529.427,Z 845.723,A -85,B 0,C 180,E1 24937.269,E2 24937.269} C_VEL
LIN {X 0,Y 529.681,Z 830.381,A -85,B 0,C 180,E1 24936.707,E2 24936.707} C_VEL
LIN {X 0,Y 529.824,Z 814.351,A -85,B 0,C 180,E1 24936.365,E2 24936.365} C_VEL
LIN {X 0,Y 530.001,Z 715.973,A -85,B 0,C 180,E1 24935.02,E2 24935.02} C_VEL
LIN {X 0,Y 529.184,Z 709.775,A -85,B 0,C 180,E1 24934.877,E2 24934.877} C_VEL
LIN {X 0,Y 529.829,Z 680.749,A -85,B 0,C 180,E1 24931.514,E2 24931.514} C_VEL
LIN {X 0,Y 530.664,Z 651.638,A -85,B 0,C 180,E1 24928.056,E2 24928.056} C_VEL
LIN {X 0,Y 531.516,Z 623.631,A -85,B 0,C 180,E1 24924.711,E2 24924.711} C_VEL
LIN {X 0,Y 532.071,Z 603.351,A -85,B 0,C 180,E1 24922.224,E2 24922.224} C_VEL
LIN {X 0,Y 528.524,Z 590.072,A -85,B 0,C 180,E1 24920.252,E2 24920.252} C_VEL
LIN {X 0,Y 528.515,Z 589.963,A -85,B 0,C 180,E1 24916.878,E2 24916.878} C_VEL
LIN {X 0,Y 528.511,Z 589.964,A -85,B 0,C 180,E1 24913.514,E2 24913.514} C_VEL
LIN {X 0,Y 528.513,Z 589.957,A -85,B 0,C 180,E1 24909.975,E2 24909.975} C_VEL
LIN {X 0,Y 528.515,Z 589.944,A -85,B 0,C 180,E1 24906.57,E2 24906.57} C_VEL
LIN {X 0,Y 528.503,Z 589.962,A -85,B 0,C 180,E1 24903.239,E2 24903.239} C_VEL
LIN {X 0,Y 528.523,Z 589.941,A -85,B 0,C 180,E1 24899.786,E2 24899.786} C_VEL
LIN {X 0,Y 528.522,Z 589.963,A -85,B 0,C 180,E1 24896.337,E2 24896.337} C_VEL
LIN {X 0,Y 528.498,Z 589.96,A -85,B 0,C 180,E1 24892.976,E2 24892.976} C_VEL
LIN {X 0,Y 528.525,Z 589.958,A -85,B 0,C 180,E1 24889.542,E2 24889.542} C_VEL
LIN {X 0,Y 528.523,Z 589.96,A -85,B 0,C 180,E1 24886.029,E2 24886.029} C_VEL
LIN {X 0,Y 528.497,Z 589.96,A -85,B 0,C 180,E1 24882.612,E2 24882.612} C_VEL
LIN {X 0,Y 528.522,Z 589.958,A -85,B 0,C 180,E1 24879.308,E2 24879.308} C_VEL
LIN {X 0,Y 528.503,Z 589.965,A -85,B 0,C 180,E1 24875.908,E2 24875.908} C_VEL
LIN {X 0,Y 528.498,Z 589.955,A -85,B 0,C 180,E1 24872.372,E2 24872.372} C_VEL
LIN {X 0,Y 528.526,Z 589.96,A -85,B 0,C 180,E1 24869.071,E2 24869.071} C_VEL
LIN {X 0,Y 528.49,Z 589.953,A -85,B 0,C 180,E1 24865.674,E2 24865.674} C_VEL
LIN {X 0,Y 528.515,Z 589.958,A -85,B 0,C 180,E1 24862.233,E2 24862.233} C_VEL
LIN {X 0,Y 528.525,Z 589.952,A -85,B 0,C 180,E1 24858.76,E2 24858.76} C_VEL
LIN {X 0,Y 528.484,Z 589.958,A -85,B 0,C 180,E1 24855.36,E2 24855.36} C_VEL
LIN {X 0,Y 528.522,Z 589.956,A -85,B 0,C 180,E1 24852.011,E2 24852.011} C_VEL
LIN {X 0,Y 528.51,Z 589.953,A -85,B 0,C 180,E1 24848.596,E2 24848.596} C_VEL
LIN {X 0,Y 528.486,Z 589.96,A -85,B 0,C 180,E1 24845.211,E2 24845.211} C_VEL
LIN {X 0,Y 528.526,Z 589.95,A -85,B 0,C 180,E1 24841.843,E2 24841.843} C_VEL
LIN {X 0,Y 528.478,Z 589.959,A -85,B 0,C 180,E1 24838.591,E2 24838.591} C_VEL
LIN {X 0,Y 528.514,Z 589.957,A -85,B 0,C 180,E1 24835.225,E2 24835.225} C_VEL
LIN {X 0,Y 528.519,Z 589.955,A -85,B 0,C 180,E1 24831.843,E2 24831.843} C_VEL
LIN {X 0,Y 528.476,Z 589.963,A -85,B 0,C 180,E1 24828.431,E2 24828.431} C_VEL
LIN {X 0,Y 528.531,Z 589.955,A -85,B 0,C 180,E1 24825.091,E2 24825.091} C_VEL
LIN {X 0,Y 528.483,Z 589.966,A -85,B 0,C 180,E1 24821.762,E2 24821.762} C_VEL
LIN {X 0,Y 528.482,Z 589.958,A -85,B 0,C 180,E1 24818.234,E2 24818.234} C_VEL
LIN {X 0,Y 528.53,Z 589.957,A -85,B 0,C 180,E1 24814.928,E2 24814.928} C_VEL
LIN {X 0,Y 528.468,Z 589.965,A -85,B 0,C 180,E1 24811.617,E2 24811.617} C_VEL
LIN {X 0,Y 528.526,Z 589.959,A -85,B 0,C 180,E1 24808.355,E2 24808.355} C_VEL
LIN {X 0,Y 528.487,Z 589.965,A -85,B 0,C 180,E1 24805.006,E2 24805.006} C_VEL
LIN {X 0,Y 528.475,Z 589.96,A -85,B 0,C 180,E1 24801.562,E2 24801.562} C_VEL
LIN {X 0,Y 528.527,Z 589.962,A -85,B 0,C 180,E1 24798.354,E2 24798.354} C_VEL
LIN {X 0,Y 528.465,Z 589.963,A -85,B 0,C 180,E1 24795.041,E2 24795.041} C_VEL
LIN {X 0,Y 528.53,Z 589.961,A -85,B 0,C 180,E1 24791.752,E2 24791.752} C_VEL
LIN {X 0,Y 528.477,Z 589.966,A -85,B 0,C 180,E1 24788.439,E2 24788.439} C_VEL
LIN {X 0,Y 528.48,Z 589.966,A -85,B 0,C 180,E1 24784.978,E2 24784.978} C_VEL
LIN {X 0,Y 528.56,Z 590.228,A -85,B 0,C 180,E1 24783.79,E2 24783.79} C_VEL
LIN {X 0,Y 535.046,Z 609.454,A -85,B 0,C 180,E1 24781.759,E2 24781.759} C_VEL
LIN {X 0,Y 533.84,Z 652.546,A -85,B 0,C 180,E1 24778.529,E2 24778.529} C_VEL
LIN {X 0,Y 532.963,Z 692.09,A -85,B 0,C 180,E1 24775.653,E2 24775.653} C_VEL
LIN {X 0,Y 534.571,Z 704.023,A -85,B 0,C 180,E1 24775.415,E2 24775.415} C_VEL
LIN {X 0,Y 533.177,Z 901.303,A -85,B 0,C 180,E1 24772.609,E2 24772.609} C_VEL
LIN {X 0,Y 532.78,Z 920.339,A -85,B 0,C 180,E1 24772.136,E2 24772.136} C_VEL
LIN {X 0,Y 532.292,Z 938.387,A -85,B 0,C 180,E1 24771.487,E2 24771.487} C_VEL
LIN {X 0,Y 531.699,Z 956.032,A -85,B 0,C 180,E1 24770.646,E2 24770.646} C_VEL
LIN {X 0,Y 531.065,Z 972.761,A -85,B 0,C 180,E1 24769.638,E2 24769.638} C_VEL
LIN {X 0,Y 530.457,Z 988.618,A -85,B 0,C 180,E1 24768.462,E2 24768.462} C_VEL
LIN {X 0,Y 529.847,Z 1003.551,A -85,B 0,C 180,E1 24767.121,E2 24767.121} C_VEL
LIN {X 0,Y 529.311,Z 1017.016,A -85,B 0,C 180,E1 24765.672,E2 24765.672} C_VEL
LIN {X 0,Y 528.854,Z 1029.275,A -85,B 0,C 180,E1 24764.097,E2 24764.097} C_VEL
LIN {X 0,Y 528.48,Z 1040.592,A -85,B 0,C 180,E1 24762.345,E2 24762.345} C_VEL
LIN {X 0,Y 528.216,Z 1050.477,A -85,B 0,C 180,E1 24760.47,E2 24760.47} C_VEL
LIN {X 0,Y 528.054,Z 1058.771,A -85,B 0,C 180,E1 24758.493,E2 24758.493} C_VEL
LIN {X 0,Y 527.964,Z 1065.109,A -85,B 0,C 180,E1 24756.525,E2 24756.525} C_VEL
LIN {X 0,Y 527.926,Z 1069.877,A -85,B 0,C 180,E1 24754.454,E2 24754.454} C_VEL
LIN {X 0,Y 527.912,Z 1072.794,A -85,B 0,C 180,E1 24752.388,E2 24752.388} C_VEL
LIN {X 0,Y 527.908,Z 1073.94,A -85,B 0,C 180,E1 24750.326,E2 24750.326} C_VEL
LIN {X 0,Y 527.912,Z 1073.346,A -85,B 0,C 180,E1 24748.264,E2 24748.264} C_VEL
LIN {X 0,Y 527.918,Z 1071.002,A -85,B 0,C 180,E1 24746.199,E2 24746.199} C_VEL
LIN {X 0,Y 527.938,Z 1067.097,A -85,B 0,C 180,E1 24744.239,E2 24744.239} C_VEL
LIN {X 0,Y 528.008,Z 1061.468,A -85,B 0,C 180,E1 24742.273,E2 24742.273} C_VEL
LIN {X 0,Y 528.127,Z 1054.428,A -85,B 0,C 180,E1 24740.41,E2 24740.41} C_VEL
LIN {X 0,Y 528.342,Z 1045.518,A -85,B 0,C 180,E1 24738.539,E2 24738.539} C_VEL
LIN {X 0,Y 528.656,Z 1035.154,A -85,B 0,C 180,E1 24736.771,E2 24736.771} C_VEL
LIN {X 0,Y 529.066,Z 1023.352,A -85,B 0,C 180,E1 24735.107,E2 24735.107} C_VEL
LIN {X 0,Y 529.608,Z 1009.573,A -85,B 0,C 180,E1 24733.493,E2 24733.493} C_VEL
LIN {X 0,Y 530.226,Z 994.544,A -85,B 0,C 180,E1 24732.037,E2 24732.037} C_VEL
LIN {X 0,Y 530.87,Z 978.439,A -85,B 0,C 180,E1 24730.756,E2 24730.756} C_VEL
LIN {X 0,Y 531.468,Z 962.26,A -85,B 0,C 180,E1 24729.702,E2 24729.702} C_VEL
LIN {X 0,Y 532.097,Z 944.809,A -85,B 0,C 180,E1 24728.794,E2 24728.794} C_VEL
LIN {X 0,Y 532.608,Z 926.534,A -85,B 0,C 180,E1 24728.063,E2 24728.063} C_VEL
LIN {X 0,Y 533.044,Z 907.982,A -85,B 0,C 180,E1 24727.535,E2 24727.535} C_VEL
LIN {X 0,Y 533.321,Z 887.491,A -85,B 0,C 180,E1 24727.171,E2 24727.171} C_VEL
LIN {X 0,Y 534.419,Z 701.292,A -85,B 0,C 180,E1 24724.54,E2 24724.54} C_VEL
LIN {X 0,Y 532.907,Z 691.327,A -85,B 0,C 180,E1 24724.316,E2 24724.316} C_VEL
LIN {X 0,Y 533.949,Z 647.689,A -85,B 0,C 180,E1 24721.11,E2 24721.11} C_VEL
LIN {X 0,Y 535.049,Z 609.065,A -85,B 0,C 180,E1 24718.213,E2 24718.213} C_VEL
LIN {X 0,Y 528.552,Z 590.187,A -85,B 0,C 180,E1 24716.206,E2 24716.206} C_VEL
LIN {X 0,Y 528.474,Z 589.968,A -85,B 0,C 180,E1 24713.012,E2 24713.012} C_VEL
LIN {X 0,Y 528.478,Z 589.967,A -85,B 0,C 180,E1 24709.514,E2 24709.514} C_VEL
LIN {X 0,Y 528.529,Z 589.959,A -85,B 0,C 180,E1 24706.18,E2 24706.18} C_VEL
LIN {X 0,Y 528.464,Z 589.967,A -85,B 0,C 180,E1 24702.928,E2 24702.928} C_VEL
LIN {X 0,Y 528.53,Z 589.965,A -85,B 0,C 180,E1 24699.608,E2 24699.608} C_VEL
LIN {X 0,Y 528.481,Z 589.963,A -85,B 0,C 180,E1 24696.296,E2 24696.296} C_VEL
LIN {X 0,Y 528.476,Z 589.965,A -85,B 0,C 180,E1 24692.856,E2 24692.856} C_VEL
LIN {X 0,Y 528.53,Z 589.96,A -85,B 0,C 180,E1 24689.587,E2 24689.587} C_VEL
LIN {X 0,Y 528.469,Z 589.965,A -85,B 0,C 180,E1 24686.259,E2 24686.259} C_VEL
LIN {X 0,Y 528.521,Z 589.96,A -85,B 0,C 180,E1 24682.882,E2 24682.882} C_VEL
LIN {X 0,Y 528.492,Z 589.958,A -85,B 0,C 180,E1 24679.564,E2 24679.564} C_VEL
LIN {X 0,Y 528.476,Z 589.964,A -85,B 0,C 180,E1 24676.148,E2 24676.148} C_VEL
LIN {X 0,Y 528.526,Z 589.957,A -85,B 0,C 180,E1 24672.899,E2 24672.899} C_VEL
LIN {X 0,Y 528.475,Z 589.956,A -85,B 0,C 180,E1 24669.584,E2 24669.584} C_VEL
LIN {X 0,Y 528.515,Z 589.963,A -85,B 0,C 180,E1 24666.19,E2 24666.19} C_VEL
LIN {X 0,Y 528.502,Z 589.96,A -85,B 0,C 180,E1 24662.819,E2 24662.819} C_VEL
LIN {X 0,Y 528.483,Z 589.961,A -85,B 0,C 180,E1 24659.458,E2 24659.458} C_VEL
LIN {X 0,Y 528.527,Z 589.962,A -85,B 0,C 180,E1 24656.095,E2 24656.095} C_VEL
LIN {X 0,Y 528.485,Z 589.962,A -85,B 0,C 180,E1 24652.717,E2 24652.717} C_VEL
LIN {X 0,Y 528.499,Z 589.965,A -85,B 0,C 180,E1 24649.205,E2 24649.205} C_VEL
LIN {X 0,Y 528.526,Z 589.954,A -85,B 0,C 180,E1 24645.875,E2 24645.875} C_VEL
LIN {X 0,Y 528.485,Z 589.959,A -85,B 0,C 180,E1 24642.466,E2 24642.466} C_VEL
LIN {X 0,Y 528.524,Z 589.961,A -85,B 0,C 180,E1 24639.05,E2 24639.05} C_VEL
LIN {X 0,Y 528.515,Z 589.956,A -85,B 0,C 180,E1 24635.643,E2 24635.643} C_VEL
LIN {X 0,Y 528.492,Z 589.964,A -85,B 0,C 180,E1 24632.263,E2 24632.263} C_VEL
LIN {X 0,Y 528.524,Z 589.965,A -85,B 0,C 180,E1 24628.905,E2 24628.905} C_VEL
LIN {X 0,Y 528.498,Z 589.963,A -85,B 0,C 180,E1 24625.55,E2 24625.55} C_VEL
LIN {X 0,Y 528.506,Z 589.967,A -85,B 0,C 180,E1 24622.058,E2 24622.058} C_VEL
LIN {X 0,Y 528.494,Z 589.966,A -85,B 0,C 180,E1 24621.718,E2 24621.718} C_VEL
LIN {X 0,Y 527.517,Z 590.265,A -85,B 0,C 180,E1 24621.144,E2 24621.144} C_VEL
LIN {X 0,Y 524.115,Z 591.922,A -85,B 0,C 180,E1 24620.303,E2 24620.303} C_VEL
LIN {X 0,Y 522.184,Z 594.178,A -85,B 0,C 180,E1 24619.718,E2 24619.718} C_VEL
LIN {X 0,Y 522.096,Z 596.525,A -85,B 0,C 180,E1 24619.299,E2 24619.299} C_VEL
LIN {X 0,Y 524.882,Z 607.148,A -85,B 0,C 180,E1 24617.744,E2 24617.744} C_VEL
LIN {X 0,Y 523.756,Z 635.103,A -85,B 0,C 180,E1 24614.284,E2 24614.284} C_VEL
LIN {X 0,Y 522.763,Z 663.459,A -85,B 0,C 180,E1 24610.853,E2 24610.853} C_VEL
LIN {X 0,Y 521.855,Z 692.663,A -85,B 0,C 180,E1 24607.332,E2 24607.332} C_VEL
LIN {X 0,Y 521.486,Z 709.755,A -85,B 0,C 180,E1 24605.351,E2 24605.351} C_VEL
LIN {X 0,Y 522.714,Z 720.22,A -85,B 0,C 180,E1 24605.13,E2 24605.13} C_VEL
LIN {X 0,Y 522.105,Z 821.962,A -85,B 0,C 180,E1 24603.666,E2 24603.666} C_VEL
LIN {X 0,Y 521.896,Z 836.894,A -85,B 0,C 180,E1 24603.243,E2 24603.243} C_VEL
LIN {X 0,Y 521.572,Z 851.636,A -85,B 0,C 180,E1 24602.594,E2 24602.594} C_VEL
LIN {X 0,Y 521.199,Z 864.972,A -85,B 0,C 180,E1 24601.776,E2 24601.776} C_VEL
LIN {X 0,Y 520.849,Z 876.759,A -85,B 0,C 180,E1 24600.834,E2 24600.834} C_VEL
LIN {X 0,Y 520.517,Z 888.902,A -85,B 0,C 180,E1 24599.582,E2 24599.582} C_VEL
LIN {X 0,Y 520.256,Z 899.311,A -85,B 0,C 180,E1 24598.215,E2 24598.215} C_VEL
LIN {X 0,Y 520.083,Z 907.293,A -85,B 0,C 180,E1 24596.858,E2 24596.858} C_VEL
LIN {X 0,Y 519.984,Z 914.095,A -85,B 0,C 180,E1 24595.344,E2 24595.344} C_VEL
LIN {X 0,Y 519.934,Z 919.321,A -85,B 0,C 180,E1 24593.698,E2 24593.698} C_VEL
LIN {X 0,Y 519.919,Z 922.567,A -85,B 0,C 180,E1 24592.025,E2 24592.025} C_VEL
LIN {X 0,Y 519.917,Z 923.897,A -85,B 0,C 180,E1 24590.488,E2 24590.488} C_VEL
LIN {X 0,Y 519.918,Z 923.508,A -85,B 0,C 180,E1 24588.733,E2 24588.733} C_VEL
LIN {X 0,Y 519.922,Z 921.277,A -85,B 0,C 180,E1 24587.101,E2 24587.101} C_VEL
LIN {X 0,Y 519.948,Z 917.315,A -85,B 0,C 180,E1 24585.503,E2 24585.503} C_VEL
LIN {X 0,Y 520.021,Z 911.404,A -85,B 0,C 180,E1 24583.907,E2 24583.907} C_VEL
LIN {X 0,Y 520.149,Z 903.892,A -85,B 0,C 180,E1 24582.433,E2 24582.433} C_VEL
LIN {X 0,Y 520.362,Z 894.919,A -85,B 0,C 180,E1 24581.078,E2 24581.078} C_VEL
LIN {X 0,Y 520.649,Z 883.975,A -85,B 0,C 180,E1 24579.785,E2 24579.785} C_VEL
LIN {X 0,Y 520.977,Z 871.936,A -85,B 0,C 180,E1 24578.665,E2 24578.665} C_VEL
LIN {X 0,Y 521.353,Z 859.401,A -85,B 0,C 180,E1 24577.77,E2 24577.77} C_VEL
LIN {X 0,Y 521.691,Z 845.99,A -85,B 0,C 180,E1 24577.046,E2 24577.046} C_VEL
LIN {X 0,Y 521.984,Z 830.857,A -85,B 0,C 180,E1 24576.475,E2 24576.475} C_VEL
LIN {X 0,Y 522.151,Z 815.082,A -85,B 0,C 180,E1 24576.126,E2 24576.126} C_VEL
LIN {X 0,Y 522.475,Z 716.903,A -85,B 0,C 180,E1 24574.737,E2 24574.737} C_VEL
LIN {X 0,Y 521.436,Z 709.646,A -85,B 0,C 180,E1 24574.57,E2 24574.57} C_VEL
LIN {X 0,Y 522.112,Z 681.907,A -85,B 0,C 180,E1 24571.317,E2 24571.317} C_VEL
LIN {X 0,Y 523.037,Z 652.754,A -85,B 0,C 180,E1 24567.809,E2 24567.809} C_VEL
LIN {X 0,Y 523.999,Z 624.761,A -85,B 0,C 180,E1 24564.415,E2 24564.415} C_VEL
LIN {X 0,Y 524.661,Z 606.197,A -85,B 0,C 180,E1 24562.113,E2 24562.113} C_VEL
LIN {X 0,Y 520.586,Z 591.052,A -85,B 0,C 180,E1 24559.85,E2 24559.85} C_VEL
LIN {X 0,Y 520.581,Z 590.948,A -85,B 0,C 180,E1 24556.335,E2 24556.335} C_VEL
LIN {X 0,Y 520.579,Z 590.951,A -85,B 0,C 180,E1 24552.91,E2 24552.91} C_VEL
LIN {X 0,Y 520.57,Z 590.95,A -85,B 0,C 180,E1 24549.421,E2 24549.421} C_VEL
LIN {X 0,Y 520.578,Z 590.927,A -85,B 0,C 180,E1 24545.972,E2 24545.972} C_VEL
LIN {X 0,Y 520.58,Z 590.952,A -85,B 0,C 180,E1 24542.543,E2 24542.543} C_VEL
LIN {X 0,Y 520.56,Z 590.931,A -85,B 0,C 180,E1 24539.147,E2 24539.147} C_VEL
LIN {X 0,Y 520.584,Z 590.947,A -85,B 0,C 180,E1 24535.678,E2 24535.678} C_VEL
LIN {X 0,Y 520.583,Z 590.949,A -85,B 0,C 180,E1 24532.129,E2 24532.129} C_VEL
LIN {X 0,Y 520.559,Z 590.951,A -85,B 0,C 180,E1 24528.79,E2 24528.79} C_VEL
LIN {X 0,Y 520.584,Z 590.946,A -85,B 0,C 180,E1 24525.287,E2 24525.287} C_VEL
LIN {X 0,Y 520.585,Z 590.943,A -85,B 0,C 180,E1 24521.795,E2 24521.795} C_VEL
LIN {X 0,Y 520.555,Z 590.95,A -85,B 0,C 180,E1 24518.346,E2 24518.346} C_VEL
LIN {X 0,Y 520.582,Z 590.939,A -85,B 0,C 180,E1 24514.902,E2 24514.902} C_VEL
LIN {X 0,Y 520.586,Z 590.953,A -85,B 0,C 180,E1 24511.366,E2 24511.366} C_VEL
LIN {X 0,Y 520.552,Z 590.949,A -85,B 0,C 180,E1 24507.925,E2 24507.925} C_VEL
LIN {X 0,Y 520.585,Z 590.942,A -85,B 0,C 180,E1 24504.511,E2 24504.511} C_VEL
LIN {X 0,Y 520.583,Z 590.953,A -85,B 0,C 180,E1 24501.021,E2 24501.021} C_VEL
LIN {X 0,Y 520.546,Z 590.939,A -85,B 0,C 180,E1 24497.552,E2 24497.552} C_VEL
LIN {X 0,Y 520.588,Z 590.946,A -85,B 0,C 180,E1 24494.118,E2 24494.118} C_VEL
LIN {X 0,Y 520.576,Z 590.946,A -85,B 0,C 180,E1 24490.626,E2 24490.626} C_VEL
LIN {X 0,Y 520.544,Z 590.944,A -85,B 0,C 180,E1 24487.172,E2 24487.172} C_VEL
LIN {X 0,Y 520.585,Z 590.945,A -85,B 0,C 180,E1 24483.744,E2 24483.744} C_VEL
LIN {X 0,Y 520.561,Z 590.942,A -85,B 0,C 180,E1 24480.33,E2 24480.33} C_VEL
LIN {X 0,Y 520.546,Z 590.95,A -85,B 0,C 180,E1 24476.917,E2 24476.917} C_VEL
LIN {X 0,Y 520.591,Z 590.937,A -85,B 0,C 180,E1 24473.494,E2 24473.494} C_VEL
LIN {X 0,Y 520.541,Z 590.952,A -85,B 0,C 180,E1 24470.157,E2 24470.157} C_VEL
LIN {X 0,Y 520.552,Z 590.944,A -85,B 0,C 180,E1 24466.674,E2 24466.674} C_VEL
LIN {X 0,Y 520.588,Z 590.953,A -85,B 0,C 180,E1 24463.371,E2 24463.371} C_VEL
LIN {X 0,Y 520.534,Z 590.949,A -85,B 0,C 180,E1 24460.007,E2 24460.007} C_VEL
LIN {X 0,Y 520.585,Z 590.948,A -85,B 0,C 180,E1 24456.647,E2 24456.647} C_VEL
LIN {X 0,Y 520.554,Z 590.948,A -85,B 0,C 180,E1 24453.273,E2 24453.273} C_VEL
LIN {X 0,Y 520.542,Z 590.949,A -85,B 0,C 180,E1 24449.912,E2 24449.912} C_VEL
LIN {X 0,Y 520.59,Z 590.95,A -85,B 0,C 180,E1 24446.549,E2 24446.549} C_VEL
LIN {X 0,Y 520.53,Z 590.955,A -85,B 0,C 180,E1 24443.226,E2 24443.226} C_VEL
LIN {X 0,Y 520.574,Z 590.951,A -85,B 0,C 180,E1 24439.857,E2 24439.857} C_VEL
LIN {X 0,Y 520.559,Z 590.957,A -85,B 0,C 180,E1 24436.556,E2 24436.556} C_VEL
LIN {X 0,Y 520.53,Z 590.952,A -85,B 0,C 180,E1 24433.12,E2 24433.12} C_VEL
LIN {X 0,Y 520.594,Z 590.952,A -85,B 0,C 180,E1 24429.804,E2 24429.804} C_VEL
LIN {X 0,Y 520.529,Z 590.955,A -85,B 0,C 180,E1 24426.546,E2 24426.546} C_VEL
LIN {X 0,Y 520.571,Z 591.184,A -85,B 0,C 180,E1 24424.264,E2 24424.264} C_VEL
LIN {X 0,Y 525.787,Z 606.256,A -85,B 0,C 180,E1 24422.603,E2 24422.603} C_VEL
LIN {X 0,Y 527.733,Z 612.347,A -85,B 0,C 180,E1 24421.975,E2 24421.975} C_VEL
LIN {X 0,Y 526.363,Z 655.035,A -85,B 0,C 180,E1 24418.724,E2 24418.724} C_VEL
LIN {X 0,Y 525.371,Z 692.306,A -85,B 0,C 180,E1 24415.959,E2 24415.959} C_VEL
LIN {X 0,Y 527.072,Z 704.989,A -85,B 0,C 180,E1 24415.705,E2 24415.705} C_VEL
LIN {X 0,Y 525.813,Z 900.219,A -85,B 0,C 180,E1 24412.966,E2 24412.966} C_VEL
LIN {X 0,Y 525.377,Z 919.575,A -85,B 0,C 180,E1 24412.491,E2 24412.491} C_VEL
LIN {X 0,Y 524.858,Z 937.086,A -85,B 0,C 180,E1 24411.866,E2 24411.866} C_VEL
LIN {X 0,Y 524.213,Z 955.025,A -85,B 0,C 180,E1 24411.013,E2 24411.013} C_VEL
LIN {X 0,Y 523.497,Z 971.947,A -85,B 0,C 180,E1 24409.992,E2 24409.992} C_VEL
LIN {X 0,Y 522.812,Z 987.983,A -85,B 0,C 180,E1 24408.796,E2 24408.796} C_VEL
LIN {X 0,Y 522.124,Z 1002.994,A -85,B 0,C 180,E1 24407.44,E2 24407.44} C_VEL
LIN {X 0,Y 521.498,Z 1017.016,A -85,B 0,C 180,E1 24405.913,E2 24405.913} C_VEL
LIN {X 0,Y 520.954,Z 1029.91,A -85,B 0,C 180,E1 24404.222,E2 24404.222} C_VEL
LIN {X 0,Y 520.537,Z 1041.226,A -85,B 0,C 180,E1 24402.424,E2 24402.424} C_VEL
LIN {X 0,Y 520.245,Z 1050.991,A -85,B 0,C 180,E1 24400.52,E2 24400.52} C_VEL
LIN {X 0,Y 520.066,Z 1059.175,A -85,B 0,C 180,E1 24398.513,E2 24398.513} C_VEL
LIN {X 0,Y 519.968,Z 1065.412,A -85,B 0,C 180,E1 24396.515,E2 24396.515} C_VEL
LIN {X 0,Y 519.927,Z 1069.877,A -85,B 0,C 180,E1 24394.522,E2 24394.522} C_VEL
LIN {X 0,Y 519.912,Z 1072.793,A -85,B 0,C 180,E1 24392.425,E2 24392.425} C_VEL
LIN {X 0,Y 519.908,Z 1073.939,A -85,B 0,C 180,E1 24390.331,E2 24390.331} C_VEL
LIN {X 0,Y 519.912,Z 1073.346,A -85,B 0,C 180,E1 24388.237,E2 24388.237} C_VEL
LIN {X 0,Y 519.916,Z 1071.161,A -85,B 0,C 180,E1 24386.251,E2 24386.251} C_VEL
LIN {X 0,Y 519.94,Z 1067.351,A -85,B 0,C 180,E1 24384.261,E2 24384.261} C_VEL
LIN {X 0,Y 520.016,Z 1061.822,A -85,B 0,C 180,E1 24382.265,E2 24382.265} C_VEL
LIN {X 0,Y 520.158,Z 1054.427,A -85,B 0,C 180,E1 24380.261,E2 24380.261} C_VEL
LIN {X 0,Y 520.402,Z 1045.517,A -85,B 0,C 180,E1 24378.361,E2 24378.361} C_VEL
LIN {X 0,Y 520.759,Z 1035.153,A -85,B 0,C 180,E1 24376.566,E2 24376.566} C_VEL
LIN {X 0,Y 521.223,Z 1023.352,A -85,B 0,C 180,E1 24374.877,E2 24374.877} C_VEL
LIN {X 0,Y 521.802,Z 1010.079,A -85,B 0,C 180,E1 24373.296,E2 24373.296} C_VEL
LIN {X 0,Y 522.483,Z 995.218,A -85,B 0,C 180,E1 24371.825,E2 24371.825} C_VEL
LIN {X 0,Y 523.203,Z 979.234,A -85,B 0,C 180,E1 24370.52,E2 24370.52} C_VEL
LIN {X 0,Y 523.916,Z 962.057,A -85,B 0,C 180,E1 24369.384,E2 24369.384} C_VEL
LIN {X 0,Y 524.623,Z 944.098,A -85,B 0,C 180,E1 24368.444,E2 24368.444} C_VEL
LIN {X 0,Y 525.182,Z 925.911,A -85,B 0,C 180,E1 24367.716,E2 24367.716} C_VEL
LIN {X 0,Y 525.65,Z 907.426,A -85,B 0,C 180,E1 24367.188,E2 24367.188} C_VEL
LIN {X 0,Y 525.954,Z 886.419,A -85,B 0,C 180,E1 24366.817,E2 24366.817} C_VEL
LIN {X 0,Y 526.882,Z 702.123,A -85,B 0,C 180,E1 24364.251,E2 24364.251} C_VEL
LIN {X 0,Y 525.304,Z 691.398,A -85,B 0,C 180,E1 24364.007,E2 24364.007} C_VEL
LIN {X 0,Y 526.498,Z 649.727,A -85,B 0,C 180,E1 24360.877,E2 24360.877} C_VEL
LIN {X 0,Y 527.741,Z 611.919,A -85,B 0,C 180,E1 24357.994,E2 24357.994} C_VEL
LIN {X 0,Y 520.593,Z 591.309,A -85,B 0,C 180,E1 24355.771,E2 24355.771} C_VEL
LIN {X 0,Y 520.551,Z 590.957,A -85,B 0,C 180,E1 24354.91,E2 24354.91} C_VEL
LIN {X 0,Y 520.532,Z 590.958,A -85,B 0,C 180,E1 24351.512,E2 24351.512} C_VEL
LIN {X 0,Y 520.592,Z 590.949,A -85,B 0,C 180,E1 24348.206,E2 24348.206} C_VEL
LIN {X 0,Y 520.527,Z 590.955,A -85,B 0,C 180,E1 24344.863,E2 24344.863} C_VEL
LIN {X 0,Y 520.565,Z 590.953,A -85,B 0,C 180,E1 24341.489,E2 24341.489} C_VEL
LIN {X 0,Y 520.558,Z 590.946,A -85,B 0,C 180,E1 24338.205,E2 24338.205} C_VEL
LIN {X 0,Y 520.529,Z 590.954,A -85,B 0,C 180,E1 24334.784,E2 24334.784} C_VEL
LIN {X 0,Y 520.593,Z 590.946,A -85,B 0,C 180,E1 24331.487,E2 24331.487} C_VEL
LIN {X 0,Y 520.535,Z 590.948,A -85,B 0,C 180,E1 24328.156,E2 24328.156} C_VEL
LIN {X 0,Y 520.551,Z 590.952,A -85,B 0,C 180,E1 24324.698,E2 24324.698} C_VEL
LIN {X 0,Y 520.586,Z 590.948,A -85,B 0,C 180,E1 24321.328,E2 24321.328} C_VEL
LIN {X 0,Y 520.534,Z 590.951,A -85,B 0,C 180,E1 24317.898,E2 24317.898} C_VEL
LIN {X 0,Y 520.576,Z 590.947,A -85,B 0,C 180,E1 24314.528,E2 24314.528} C_VEL
LIN {X 0,Y 520.559,Z 590.95,A -85,B 0,C 180,E1 24311.186,E2 24311.186} C_VEL
LIN {X 0,Y 520.54,Z 590.954,A -85,B 0,C 180,E1 24307.727,E2 24307.727} C_VEL
LIN {X 0,Y 520.587,Z 590.944,A -85,B 0,C 180,E1 24304.406,E2 24304.406} C_VEL
LIN {X 0,Y 520.546,Z 590.949,A -85,B 0,C 180,E1 24300.99,E2 24300.99} C_VEL
LIN {X 0,Y 520.551,Z 590.954,A -85,B 0,C 180,E1 24297.468,E2 24297.468} C_VEL
LIN {X 0,Y 520.588,Z 590.945,A -85,B 0,C 180,E1 24294.047,E2 24294.047} C_VEL
LIN {X 0,Y 520.545,Z 590.944,A -85,B 0,C 180,E1 24290.715,E2 24290.715} C_VEL
LIN {X 0,Y 520.567,Z 590.948,A -85,B 0,C 180,E1 24287.239,E2 24287.239} C_VEL
LIN {X 0,Y 520.588,Z 590.95,A -85,B 0,C 180,E1 24283.805,E2 24283.805} C_VEL
LIN {X 0,Y 520.549,Z 590.951,A -85,B 0,C 180,E1 24280.358,E2 24280.358} C_VEL
LIN {X 0,Y 520.581,Z 590.95,A -85,B 0,C 180,E1 24276.926,E2 24276.926} C_VEL
LIN {X 0,Y 520.587,Z 590.95,A -85,B 0,C 180,E1 24273.416,E2 24273.416} C_VEL
LIN {X 0,Y 520.552,Z 590.953,A -85,B 0,C 180,E1 24270.028,E2 24270.028} C_VEL
LIN {X 0,Y 520.587,Z 590.952,A -85,B 0,C 180,E1 24266.666,E2 24266.666} C_VEL
LIN {X 0,Y 520.578,Z 590.953,A -85,B 0,C 180,E1 24263.183,E2 24263.183} C_VEL
LIN {X 0,Y 520.615,Z 591.211,A -85,B 0,C 180,E1 24260.108,E2 24260.108} C_VEL
LIN {X 0,Y 522.096,Z 596.525,A -85,B 0,C 180,E1 24259.299,E2 24259.299} C_VEL
LIN {X 0,Y 522.435,Z 600.714,A -85,B 0,C 180,E1 24258.734,E2 24258.734} C_VEL
LIN {X 0,Y 520.998,Z 606.863,A -85,B 0,C 180,E1 24258.038,E2 24258.038} C_VEL
LIN {X 0,Y 517.31,Z 618.012,A -85,B 0,C 180,E1 24256.841,E2 24256.841} C_VEL
LIN {X 0,Y 516.886,Z 621.095,A -85,B 0,C 180,E1 24256.471,E2 24256.471} C_VEL
LIN {X 0,Y 515.703,Z 649.366,A -85,B 0,C 180,E1 24252.961,E2 24252.961} C_VEL
LIN {X 0,Y 514.666,Z 678.121,A -85,B 0,C 180,E1 24249.44,E2 24249.44} C_VEL
LIN {X 0,Y 513.756,Z 707.835,A -85,B 0,C 180,E1 24245.859,E2 24245.859} C_VEL
LIN {X 0,Y 513.829,Z 710.061,A -85,B 0,C 180,E1 24245.667,E2 24245.667} C_VEL
LIN {X 0,Y 515.234,Z 721.002,A -85,B 0,C 180,E1 24245.435,E2 24245.435} C_VEL
LIN {X 0,Y 514.535,Z 822.63,A -85,B 0,C 180,E1 24243.943,E2 24243.943} C_VEL
LIN {X 0,Y 514.309,Z 837.621,A -85,B 0,C 180,E1 24243.512,E2 24243.512} C_VEL
LIN {X 0,Y 513.967,Z 852.016,A -85,B 0,C 180,E1 24242.872,E2 24242.872} C_VEL
LIN {X 0,Y 513.588,Z 864.598,A -85,B 0,C 180,E1 24242.105,E2 24242.105} C_VEL
LIN {X 0,Y 513.167,Z 877.391,A -85,B 0,C 180,E1 24241.086,E2 24241.086} C_VEL
LIN {X 0,Y 512.795,Z 889.009,A -85,B 0,C 180,E1 24239.88,E2 24239.88} C_VEL
LIN {X 0,Y 512.457,Z 898.661,A -85,B 0,C 180,E1 24238.597,E2 24238.597} C_VEL
LIN {X 0,Y 512.201,Z 907.006,A -85,B 0,C 180,E1 24237.18,E2 24237.18} C_VEL
LIN {X 0,Y 512.035,Z 914.174,A -85,B 0,C 180,E1 24235.556,E2 24235.556} C_VEL
LIN {X 0,Y 511.951,Z 919.446,A -85,B 0,C 180,E1 24233.846,E2 24233.846} C_VEL
LIN {X 0,Y 511.925,Z 922.587,A -85,B 0,C 180,E1 24232.212,E2 24232.212} C_VEL
LIN {X 0,Y 511.919,Z 924.059,A -85,B 0,C 180,E1 24230.583,E2 24230.583} C_VEL
LIN {X 0,Y 511.92,Z 923.754,A -85,B 0,C 180,E1 24228.8,E2 24228.8} C_VEL
LIN {X 0,Y 511.927,Z 921.716,A -85,B 0,C 180,E1 24227.153,E2 24227.153} C_VEL
LIN {X 0,Y 511.969,Z 917.976,A -85,B 0,C 180,E1 24225.519,E2 24225.519} C_VEL
LIN {X 0,Y 512.067,Z 912.329,A -85,B 0,C 180,E1 24223.896,E2 24223.896} C_VEL
LIN {X 0,Y 512.24,Z 905.165,A -85,B 0,C 180,E1 24222.399,E2 24222.399} C_VEL
LIN {X 0,Y 512.514,Z 896.599,A -85,B 0,C 180,E1 24221.022,E2 24221.022} C_VEL
LIN {X 0,Y 512.868,Z 886.054,A -85,B 0,C 180,E1 24219.708,E2 24219.708} C_VEL
LIN {X 0,Y 513.203,Z 874.974,A -85,B 0,C 180,E1 24218.628,E2 24218.628} C_VEL
LIN {X 0,Y 513.609,Z 863.145,A -85,B 0,C 180,E1 24217.719,E2 24217.719} C_VEL
LIN {X 0,Y 513.989,Z 849.513,A -85,B 0,C 180,E1 24216.927,E2 24216.927} C_VEL
LIN {X 0,Y 514.302,Z 835.404,A -85,B 0,C 180,E1 24216.338,E2 24216.338} C_VEL
LIN {X 0,Y 514.522,Z 820.262,A -85,B 0,C 180,E1 24215.932,E2 24215.932} C_VEL
LIN {X 0,Y 514.952,Z 717.759,A -85,B 0,C 180,E1 24214.444,E2 24214.444} C_VEL
LIN {X 0,Y 513.683,Z 709.28,A -85,B 0,C 180,E1 24214.235,E2 24214.235} C_VEL
LIN {X 0,Y 514.43,Z 682.149,A -85,B 0,C 180,E1 24211.002,E2 24211.002} C_VEL
LIN {X 0,Y 515.42,Z 653.87,A -85,B 0,C 180,E1 24207.554,E2 24207.554} C_VEL
LIN {X 0,Y 516.495,Z 625.892,A -85,B 0,C 180,E1 24204.111,E2 24204.111} C_VEL
LIN {X 0,Y 517.087,Z 608.381,A -85,B 0,C 180,E1 24201.902,E2 24201.902} C_VEL
LIN {X 0,Y 512.655,Z 592.03,A -85,B 0,C 180,E1 24199.436,E2 24199.436} C_VEL
LIN {X 0,Y 512.629,Z 591.94,A -85,B 0,C 180,E1 24195.888,E2 24195.888} C_VEL
LIN {X 0,Y 512.644,Z 591.935,A -85,B 0,C 180,E1 24192.403,E2 24192.403} C_VEL
LIN {X 0,Y 512.644,Z 591.942,A -85,B 0,C 180,E1 24188.849,E2 24188.849} C_VEL
LIN {X 0,Y 512.623,Z 591.921,A -85,B 0,C 180,E1 24185.358,E2 24185.358} C_VEL
LIN {X 0,Y 512.647,Z 591.934,A -85,B 0,C 180,E1 24181.834,E2 24181.834} C_VEL
LIN {X 0,Y 512.64,Z 591.921,A -85,B 0,C 180,E1 24178.354,E2 24178.354} C_VEL
LIN {X 0,Y 512.626,Z 591.941,A -85,B 0,C 180,E1 24174.873,E2 24174.873} C_VEL
LIN {X 0,Y 512.64,Z 591.934,A -85,B 0,C 180,E1 24171.381,E2 24171.381} C_VEL
LIN {X 0,Y 512.644,Z 591.932,A -85,B 0,C 180,E1 24167.86,E2 24167.86} C_VEL
LIN {X 0,Y 512.623,Z 591.94,A -85,B 0,C 180,E1 24164.445,E2 24164.445} C_VEL
LIN {X 0,Y 512.637,Z 591.924,A -85,B 0,C 180,E1 24160.946,E2 24160.946} C_VEL
LIN {X 0,Y 512.647,Z 591.94,A -85,B 0,C 180,E1 24157.456,E2 24157.456} C_VEL
LIN {X 0,Y 512.617,Z 591.933,A -85,B 0,C 180,E1 24154.007,E2 24154.007} C_VEL
LIN {X 0,Y 512.63,Z 591.937,A -85,B 0,C 180,E1 24150.446,E2 24150.446} C_VEL
LIN {X 0,Y 512.648,Z 591.926,A -85,B 0,C 180,E1 24146.959,E2 24146.959} C_VEL
LIN {X 0,Y 512.613,Z 591.937,A -85,B 0,C 180,E1 24143.544,E2 24143.544} C_VEL
LIN {X 0,Y 512.63,Z 591.934,A -85,B 0,C 180,E1 24140.077,E2 24140.077} C_VEL
LIN {X 0,Y 512.646,Z 591.93,A -85,B 0,C 180,E1 24136.661,E2 24136.661} C_VEL
LIN {X 0,Y 512.607,Z 591.941,A -85,B 0,C 180,E1 24133.263,E2 24133.263} C_VEL
LIN {X 0,Y 512.633,Z 591.924,A -85,B 0,C 180,E1 24129.77,E2 24129.77} C_VEL
LIN {X 0,Y 512.651,Z 591.94,A -85,B 0,C 180,E1 24126.271,E2 24126.271} C_VEL
LIN {X 0,Y 512.604,Z 591.94,A -85,B 0,C 180,E1 24122.795,E2 24122.795} C_VEL
LIN {X 0,Y 512.631,Z 591.93,A -85,B 0,C 180,E1 24119.33,E2 24119.33} C_VEL
LIN {X 0,Y 512.648,Z 591.94,A -85,B 0,C 180,E1 24115.862,E2 24115.862} C_VEL
LIN {X 0,Y 512.597,Z 591.929,A -85,B 0,C 180,E1 24112.491,E2 24112.491} C_VEL
LIN {X 0,Y 512.642,Z 591.937,A -85,B 0,C 180,E1 24109.095,E2 24109.095} C_VEL
LIN {X 0,Y 512.629,Z 591.934,A -85,B 0,C 180,E1 24105.658,E2 24105.658} C_VEL
LIN {X 0,Y 512.6,Z 591.941,A -85,B 0,C 180,E1 24102.285,E2 24102.285} C_VEL
LIN {X 0,Y 512.653,Z 591.933,A -85,B 0,C 180,E1 24098.85,E2 24098.85} C_VEL
LIN {X 0,Y 512.609,Z 591.945,A -85,B 0,C 180,E1 24095.452,E2 24095.452} C_VEL
LIN {X 0,Y 512.601,Z 591.941,A -85,B 0,C 180,E1 24091.96,E2 24091.96} C_VEL
LIN {X 0,Y 512.654,Z 591.937,A -85,B 0,C 180,E1 24088.618,E2 24088.618} C_VEL
LIN {X 0,Y 512.591,Z 591.942,A -85,B 0,C 180,E1 24085.28,E2 24085.28} C_VEL
LIN {X 0,Y 512.621,Z 591.935,A -85,B 0,C 180,E1 24081.808,E2 24081.808} C_VEL
LIN {X 0,Y 512.639,Z 591.94,A -85,B 0,C 180,E1 24078.46,E2 24078.46} C_VEL
LIN {X 0,Y 512.589,Z 591.941,A -85,B 0,C 180,E1 24075.079,E2 24075.079} C_VEL
LIN {X 0,Y 512.65,Z 591.939,A -85,B 0,C 180,E1 24071.67,E2 24071.67} C_VEL
LIN {X 0,Y 512.606,Z 591.943,A -85,B 0,C 180,E1 24068.337,E2 24068.337} C_VEL
LIN {X 0,Y 512.603,Z 592.008,A -85,B 0,C 180,E1 24064.856,E2 24064.856} C_VEL
LIN {X 0,Y 512.666,Z 592.44,A -85,B 0,C 180,E1 24064.678,E2 24064.678} C_VEL
LIN {X 0,Y 520.441,Z 614.923,A -85,B 0,C 180,E1 24062.224,E2 24062.224} C_VEL
LIN {X 0,Y 518.981,Z 654.284,A -85,B 0,C 180,E1 24059.172,E2 24059.172} C_VEL
LIN {X 0,Y 517.799,Z 692.48,A -85,B 0,C 180,E1 24056.275,E2 24056.275} C_VEL
LIN {X 0,Y 519.579,Z 705.972,A -85,B 0,C 180,E1 24056.002,E2 24056.002} C_VEL
LIN {X 0,Y 518.219,Z 900.863,A -85,B 0,C 180,E1 24053.235,E2 24053.235} C_VEL
LIN {X 0,Y 517.77,Z 920.186,A -85,B 0,C 180,E1 24052.755,E2 24052.755} C_VEL
LIN {X 0,Y 517.216,Z 938.688,A -85,B 0,C 180,E1 24052.086,E2 24052.086} C_VEL
LIN {X 0,Y 516.562,Z 956.745,A -85,B 0,C 180,E1 24051.221,E2 24051.221} C_VEL
LIN {X 0,Y 515.864,Z 972.755,A -85,B 0,C 180,E1 24050.242,E2 24050.242} C_VEL
LIN {X 0,Y 515.113,Z 988.614,A -85,B 0,C 180,E1 24049.032,E2 24049.032} C_VEL
LIN {X 0,Y 514.356,Z 1003.548,A -85,B 0,C 180,E1 24047.653,E2 24047.653} C_VEL
LIN {X 0,Y 513.69,Z 1017.016,A -85,B 0,C 180,E1 24046.161,E2 24046.161} C_VEL
LIN {X 0,Y 513.086,Z 1029.909,A -85,B 0,C 180,E1 24044.444,E2 24044.444} C_VEL
LIN {X 0,Y 512.622,Z 1041.225,A -85,B 0,C 180,E1 24042.619,E2 24042.619} C_VEL
LIN {X 0,Y 512.292,Z 1050.991,A -85,B 0,C 180,E1 24040.686,E2 24040.686} C_VEL
LIN {X 0,Y 512.086,Z 1059.175,A -85,B 0,C 180,E1 24038.647,E2 24038.647} C_VEL
LIN {X 0,Y 511.975,Z 1065.412,A -85,B 0,C 180,E1 24036.617,E2 24036.617} C_VEL
LIN {X 0,Y 511.928,Z 1069.876,A -85,B 0,C 180,E1 24034.593,E2 24034.593} C_VEL
LIN {X 0,Y 511.911,Z 1072.793,A -85,B 0,C 180,E1 24032.463,E2 24032.463} C_VEL
LIN {X 0,Y 511.908,Z 1073.939,A -85,B 0,C 180,E1 24030.336,E2 24030.336} C_VEL
LIN {X 0,Y 511.912,Z 1073.414,A -85,B 0,C 180,E1 24028.321,E2 24028.321} C_VEL
LIN {X 0,Y 511.918,Z 1071.16,A -85,B 0,C 180,E1 24026.193,E2 24026.193} C_VEL
LIN {X 0,Y 511.944,Z 1067.351,A -85,B 0,C 180,E1 24024.171,E2 24024.171} C_VEL
LIN {X 0,Y 512.029,Z 1061.822,A -85,B 0,C 180,E1 24022.144,E2 24022.144} C_VEL
LIN {X 0,Y 512.195,Z 1054.427,A -85,B 0,C 180,E1 24020.109,E2 24020.109} C_VEL
LIN {X 0,Y 512.467,Z 1045.517,A -85,B 0,C 180,E1 24018.179,E2 24018.179} C_VEL
LIN {X 0,Y 512.865,Z 1035.152,A -85,B 0,C 180,E1 24016.356,E2 24016.356} C_VEL
LIN {X 0,Y 513.409,Z 1022.907,A -85,B 0,C 180,E1 24014.581,E2 24014.581} C_VEL
LIN {X 0,Y 514.082,Z 1009.064,A -85,B 0,C 180,E1 24012.921,E2 24012.921} C_VEL
LIN {X 0,Y 514.845,Z 993.958,A -85,B 0,C 180,E1 24011.428,E2 24011.428} C_VEL
LIN {X 0,Y 515.625,Z 978.003,A -85,B 0,C 180,E1 24010.131,E2 24010.131} C_VEL
LIN {X 0,Y 516.355,Z 961.913,A -85,B 0,C 180,E1 24009.068,E2 24009.068} C_VEL
LIN {X 0,Y 517.034,Z 944.364,A -85,B 0,C 180,E1 24008.162,E2 24008.162} C_VEL
LIN {X 0,Y 517.593,Z 925.907,A -85,B 0,C 180,E1 24007.432,E2 24007.432} C_VEL
LIN {X 0,Y 518.062,Z 907.072,A -85,B 0,C 180,E1 24006.9,E2 24006.9} C_VEL
LIN {X 0,Y 518.367,Z 885.778,A -85,B 0,C 180,E1 24006.53,E2 24006.53} C_VEL
LIN {X 0,Y 519.38,Z 703.119,A -85,B 0,C 180,E1 24003.959,E2 24003.959} C_VEL
LIN {X 0,Y 517.722,Z 691.742,A -85,B 0,C 180,E1 24003.706,E2 24003.706} C_VEL
LIN {X 0,Y 519.154,Z 648.615,A -85,B 0,C 180,E1 24000.396,E2 24000.396} C_VEL
LIN {X 0,Y 520.411,Z 614.517,A -85,B 0,C 180,E1 23997.745,E2 23997.745} C_VEL
LIN {X 0,Y 513.142,Z 594.039,A -85,B 0,C 180,E1 23995.509,E2 23995.509} C_VEL
LIN {X 0,Y 512.616,Z 592.14,A -85,B 0,C 180,E1 23995.247,E2 23995.247} C_VEL
LIN {X 0,Y 512.634,Z 591.943,A -85,B 0,C 180,E1 23991.951,E2 23991.951} C_VEL
LIN {X 0,Y 512.616,Z 591.94,A -85,B 0,C 180,E1 23988.607,E2 23988.607} C_VEL
LIN {X 0,Y 512.591,Z 591.946,A -85,B 0,C 180,E1 23985.236,E2 23985.236} C_VEL
LIN {X 0,Y 512.649,Z 591.941,A -85,B 0,C 180,E1 23981.988,E2 23981.988} C_VEL
LIN {X 0,Y 512.585,Z 591.939,A -85,B 0,C 180,E1 23978.717,E2 23978.717} C_VEL
LIN {X 0,Y 512.641,Z 591.938,A -85,B 0,C 180,E1 23975.386,E2 23975.386} C_VEL
LIN {X 0,Y 512.613,Z 591.938,A -85,B 0,C 180,E1 23972.042,E2 23972.042} C_VEL
LIN {X 0,Y 512.594,Z 591.94,A -85,B 0,C 180,E1 23968.626,E2 23968.626} C_VEL
LIN {X 0,Y 512.651,Z 591.94,A -85,B 0,C 180,E1 23965.285,E2 23965.285} C_VEL
LIN {X 0,Y 512.599,Z 591.941,A -85,B 0,C 180,E1 23961.873,E2 23961.873} C_VEL
LIN {X 0,Y 512.602,Z 591.943,A -85,B 0,C 180,E1 23958.303,E2 23958.303} C_VEL
LIN {X 0,Y 512.653,Z 591.936,A -85,B 0,C 180,E1 23954.918,E2 23954.918} C_VEL
LIN {X 0,Y 512.602,Z 591.941,A -85,B 0,C 180,E1 23951.476,E2 23951.476} C_VEL
LIN {X 0,Y 512.612,Z 591.944,A -85,B 0,C 180,E1 23947.96,E2 23947.96} C_VEL
LIN {X 0,Y 512.646,Z 591.932,A -85,B 0,C 180,E1 23944.586,E2 23944.586} C_VEL
LIN {X 0,Y 512.6,Z 591.939,A -85,B 0,C 180,E1 23941.229,E2 23941.229} C_VEL
LIN {X 0,Y 512.633,Z 591.945,A -85,B 0,C 180,E1 23937.764,E2 23937.764} C_VEL
LIN {X 0,Y 512.641,Z 591.932,A -85,B 0,C 180,E1 23934.291,E2 23934.291} C_VEL
LIN {X 0,Y 512.604,Z 591.933,A -85,B 0,C 180,E1 23930.909,E2 23930.909} C_VEL
LIN {X 0,Y 512.646,Z 591.938,A -85,B 0,C 180,E1 23927.497,E2 23927.497} C_VEL
LIN {X 0,Y 512.632,Z 591.939,A -85,B 0,C 180,E1 23924.037,E2 23924.037} C_VEL
LIN {X 0,Y 512.61,Z 591.941,A -85,B 0,C 180,E1 23920.516,E2 23920.516} C_VEL
LIN {X 0,Y 512.648,Z 591.943,A -85,B 0,C 180,E1 23917.162,E2 23917.162} C_VEL
LIN {X 0,Y 512.629,Z 591.939,A -85,B 0,C 180,E1 23913.72,E2 23913.72} C_VEL
LIN {X 0,Y 512.616,Z 591.942,A -85,B 0,C 180,E1 23910.173,E2 23910.173} C_VEL
LIN {X 0,Y 512.648,Z 591.942,A -85,B 0,C 180,E1 23906.766,E2 23906.766} C_VEL
LIN {X 0,Y 512.632,Z 591.943,A -85,B 0,C 180,E1 23903.286,E2 23903.286} C_VEL
LIN {X 0,Y 512.684,Z 592.208,A -85,B 0,C 180,E1 23900.554,E2 23900.554} C_VEL
LIN {X 0,Y 517.378,Z 609.292,A -85,B 0,C 180,E1 23897.961,E2 23897.961} C_VEL
LIN {X 0,Y 516.886,Z 621.095,A -85,B 0,C 180,E1 23896.471,E2 23896.471} C_VEL
LIN {X 0,Y 515.725,Z 626.446,A -85,B 0,C 180,E1 23895.86,E2 23895.86} C_VEL
LIN {X 0,Y 509.012,Z 642.219,A -85,B 0,C 180,E1 23894.249,E2 23894.249} C_VEL
LIN {X 0,Y 508.345,Z 646.04,A -85,B 0,C 180,E1 23893.799,E2 23893.799} C_VEL
LIN {X 0,Y 507.147,Z 675.501,A -85,B 0,C 180,E1 23890.143,E2 23890.143} C_VEL
LIN {X 0,Y 506.111,Z 705.367,A -85,B 0,C 180,E1 23886.487,E2 23886.487} C_VEL
LIN {X 0,Y 506.075,Z 709.586,A -85,B 0,C 180,E1 23886.02,E2 23886.02} C_VEL
LIN {X 0,Y 507.77,Z 721.423,A -85,B 0,C 180,E1 23885.755,E2 23885.755} C_VEL
LIN {X 0,Y 506.975,Z 823.364,A -85,B 0,C 180,E1 23884.228,E2 23884.228} C_VEL
LIN {X 0,Y 506.745,Z 837.836,A -85,B 0,C 180,E1 23883.808,E2 23883.808} C_VEL
LIN {X 0,Y 506.372,Z 852.5,A -85,B 0,C 180,E1 23883.152,E2 23883.152} C_VEL
LIN {X 0,Y 505.963,Z 865.121,A -85,B 0,C 180,E1 23882.38,E2 23882.38} C_VEL
LIN {X 0,Y 505.496,Z 878.009,A -85,B 0,C 180,E1 23881.346,E2 23881.346} C_VEL
LIN {X 0,Y 505.093,Z 889.155,A -85,B 0,C 180,E1 23880.186,E2 23880.186} C_VEL
LIN {X 0,Y 504.706,Z 899.065,A -85,B 0,C 180,E1 23878.879,E2 23878.879} C_VEL
LIN {X 0,Y 504.388,Z 907.953,A -85,B 0,C 180,E1 23877.366,E2 23877.366} C_VEL
LIN {X 0,Y 504.181,Z 915.073,A -85,B 0,C 180,E1 23875.741,E2 23875.741} C_VEL
LIN {X 0,Y 504.071,Z 920.142,A -85,B 0,C 180,E1 23874.118,E2 23874.118} C_VEL
LIN {X 0,Y 504.025,Z 923.57,A -85,B 0,C 180,E1 23872.417,E2 23872.417} C_VEL
LIN {X 0,Y 504.01,Z 925.215,A -85,B 0,C 180,E1 23870.678,E2 23870.678} C_VEL
LIN {X 0,Y 504.01,Z 925.063,A -85,B 0,C 180,E1 23868.986,E2 23868.986} C_VEL
LIN {X 0,Y 504.023,Z 923.264,A -85,B 0,C 180,E1 23867.311,E2 23867.311} C_VEL
LIN {X 0,Y 504.076,Z 919.404,A -85,B 0,C 180,E1 23865.532,E2 23865.532} C_VEL
LIN {X 0,Y 504.195,Z 913.866,A -85,B 0,C 180,E1 23863.884,E2 23863.884} C_VEL
LIN {X 0,Y 504.394,Z 906.856,A -85,B 0,C 180,E1 23862.362,E2 23862.362} C_VEL
LIN {X 0,Y 504.694,Z 898.443,A -85,B 0,C 180,E1 23860.964,E2 23860.964} C_VEL
LIN {X 0,Y 505.079,Z 888.277,A -85,B 0,C 180,E1 23859.649,E2 23859.649} C_VEL
LIN {X 0,Y 505.456,Z 877.349,A -85,B 0,C 180,E1 23858.532,E2 23858.532} C_VEL
LIN {X 0,Y 505.94,Z 864.233,A -85,B 0,C 180,E1 23857.494,E2 23857.494} C_VEL
LIN {X 0,Y 506.363,Z 850.35,A -85,B 0,C 180,E1 23856.673,E2 23856.673} C_VEL
LIN {X 0,Y 506.698,Z 836.262,A -85,B 0,C 180,E1 23856.074,E2 23856.074} C_VEL
LIN {X 0,Y 506.937,Z 820.863,A -85,B 0,C 180,E1 23855.654,E2 23855.654} C_VEL
LIN {X 0,Y 507.445,Z 718.632,A -85,B 0,C 180,E1 23854.142,E2 23854.142} C_VEL
LIN {X 0,Y 505.956,Z 709.092,A -85,B 0,C 180,E1 23853.902,E2 23853.902} C_VEL
LIN {X 0,Y 506.838,Z 680.56,A -85,B 0,C 180,E1 23850.452,E2 23850.452} C_VEL
LIN {X 0,Y 507.931,Z 652.247,A -85,B 0,C 180,E1 23846.953,E2 23846.953} C_VEL
LIN {X 0,Y 509.183,Z 623.435,A -85,B 0,C 180,E1 23843.347,E2 23843.347} C_VEL
LIN {X 0,Y 509.637,Z 611.076,A -85,B 0,C 180,E1 23841.766,E2 23841.766} C_VEL
LIN {X 0,Y 504.714,Z 593.057,A -85,B 0,C 180,E1 23839.036,E2 23839.036} C_VEL
LIN {X 0,Y 504.701,Z 592.931,A -85,B 0,C 180,E1 23835.545,E2 23835.545} C_VEL
LIN {X 0,Y 504.695,Z 592.926,A -85,B 0,C 180,E1 23831.979,E2 23831.979} C_VEL
LIN {X 0,Y 504.702,Z 592.927,A -85,B 0,C 180,E1 23828.5,E2 23828.5} C_VEL
LIN {X 0,Y 504.702,Z 592.913,A -85,B 0,C 180,E1 23824.915,E2 23824.915} C_VEL
LIN {X 0,Y 504.686,Z 592.927,A -85,B 0,C 180,E1 23821.361,E2 23821.361} C_VEL
LIN {X 0,Y 504.704,Z 592.914,A -85,B 0,C 180,E1 23817.931,E2 23817.931} C_VEL
LIN {X 0,Y 504.705,Z 592.931,A -85,B 0,C 180,E1 23814.377,E2 23814.377} C_VEL
LIN {X 0,Y 504.683,Z 592.926,A -85,B 0,C 180,E1 23810.949,E2 23810.949} C_VEL
LIN {X 0,Y 504.704,Z 592.916,A -85,B 0,C 180,E1 23807.474,E2 23807.474} C_VEL
LIN {X 0,Y 504.706,Z 592.931,A -85,B 0,C 180,E1 23803.898,E2 23803.898} C_VEL
LIN {X 0,Y 504.678,Z 592.917,A -85,B 0,C 180,E1 23800.38,E2 23800.38} C_VEL
LIN {X 0,Y 504.702,Z 592.924,A -85,B 0,C 180,E1 23796.89,E2 23796.89} C_VEL
LIN {X 0,Y 504.71,Z 592.918,A -85,B 0,C 180,E1 23793.418,E2 23793.418} C_VEL
LIN {X 0,Y 504.674,Z 592.93,A -85,B 0,C 180,E1 23789.952,E2 23789.952} C_VEL
LIN {X 0,Y 504.701,Z 592.911,A -85,B 0,C 180,E1 23786.471,E2 23786.471} C_VEL
LIN {X 0,Y 504.71,Z 592.93,A -85,B 0,C 180,E1 23782.898,E2 23782.898} C_VEL
LIN {X 0,Y 504.672,Z 592.928,A -85,B 0,C 180,E1 23779.428,E2 23779.428} C_VEL
LIN {X 0,Y 504.686,Z 592.92,A -85,B 0,C 180,E1 23775.867,E2 23775.867} C_VEL
LIN {X 0,Y 504.712,Z 592.926,A -85,B 0,C 180,E1 23772.401,E2 23772.401} C_VEL
LIN {X 0,Y 504.668,Z 592.918,A -85,B 0,C 180,E1 23769.005,E2 23769.005} C_VEL
LIN {X 0,Y 504.693,Z 592.924,A -85,B 0,C 180,E1 23765.571,E2 23765.571} C_VEL
LIN {X 0,Y 504.708,Z 592.917,A -85,B 0,C 180,E1 23762.044,E2 23762.044} C_VEL
LIN {X 0,Y 504.661,Z 592.924,A -85,B 0,C 180,E1 23758.638,E2 23758.638} C_VEL
LIN {X 0,Y 504.686,Z 592.924,A -85,B 0,C 180,E1 23755.113,E2 23755.113} C_VEL
LIN {X 0,Y 504.712,Z 592.92,A -85,B 0,C 180,E1 23751.685,E2 23751.685} C_VEL
LIN {X 0,Y 504.659,Z 592.931,A -85,B 0,C 180,E1 23748.341,E2 23748.341} C_VEL
LIN {X 0,Y 504.709,Z 592.92,A -85,B 0,C 180,E1 23744.959,E2 23744.959} C_VEL
LIN {X 0,Y 504.689,Z 592.934,A -85,B 0,C 180,E1 23741.52,E2 23741.52} C_VEL
LIN {X 0,Y 504.66,Z 592.926,A -85,B 0,C 180,E1 23738.132,E2 23738.132} C_VEL
LIN {X 0,Y 504.713,Z 592.92,A -85,B 0,C 180,E1 23734.791,E2 23734.791} C_VEL
LIN {X 0,Y 504.657,Z 592.933,A -85,B 0,C 180,E1 23731.479,E2 23731.479} C_VEL
LIN {X 0,Y 504.676,Z 592.928,A -85,B 0,C 180,E1 23727.99,E2 23727.99} C_VEL
LIN {X 0,Y 504.711,Z 592.927,A -85,B 0,C 180,E1 23724.518,E2 23724.518} C_VEL
LIN {X 0,Y 504.651,Z 592.929,A -85,B 0,C 180,E1 23721.138,E2 23721.138} C_VEL
LIN {X 0,Y 504.696,Z 592.928,A -85,B 0,C 180,E1 23717.81,E2 23717.81} C_VEL
LIN {X 0,Y 504.689,Z 592.933,A -85,B 0,C 180,E1 23714.375,E2 23714.375} C_VEL
LIN {X 0,Y 504.65,Z 592.933,A -85,B 0,C 180,E1 23710.982,E2 23710.982} C_VEL
LIN {X 0,Y 504.716,Z 592.93,A -85,B 0,C 180,E1 23707.745,E2 23707.745} C_VEL
LIN {X 0,Y 504.719,Z 593.172,A -85,B 0,C 180,E1 23705.204,E2 23705.204} C_VEL
LIN {X 0,Y 512.423,Z 615.276,A -85,B 0,C 180,E1 23702.718,E2 23702.718} C_VEL
LIN {X 0,Y 513.151,Z 617.635,A -85,B 0,C 180,E1 23702.469,E2 23702.469} C_VEL
LIN {X 0,Y 511.743,Z 650.291,A -85,B 0,C 180,E1 23699.883,E2 23699.883} C_VEL
LIN {X 0,Y 510.22,Z 692.426,A -85,B 0,C 180,E1 23696.608,E2 23696.608} C_VEL
LIN {X 0,Y 512.102,Z 707.006,A -85,B 0,C 180,E1 23696.307,E2 23696.307} C_VEL
LIN {X 0,Y 510.627,Z 900.319,A -85,B 0,C 180,E1 23693.525,E2 23693.525} C_VEL
LIN {X 0,Y 510.138,Z 919.528,A -85,B 0,C 180,E1 23693.041,E2 23693.041} C_VEL
LIN {X 0,Y 509.546,Z 937.735,A -85,B 0,C 180,E1 23692.376,E2 23692.376} C_VEL
LIN {X 0,Y 508.848,Z 955.825,A -85,B 0,C 180,E1 23691.498,E2 23691.498} C_VEL
LIN {X 0,Y 508.066,Z 972.97,A -85,B 0,C 180,E1 23690.446,E2 23690.446} C_VEL
LIN {X 0,Y 507.31,Z 989.252,A -85,B 0,C 180,E1 23689.217,E2 23689.217} C_VEL
LIN {X 0,Y 506.552,Z 1004.56,A -85,B 0,C 180,E1 23687.815,E2 23687.815} C_VEL
LIN {X 0,Y 505.89,Z 1017.016,A -85,B 0,C 180,E1 23686.418,E2 23686.418} C_VEL
LIN {X 0,Y 505.227,Z 1029.908,A -85,B 0,C 180,E1 23684.674,E2 23684.674} C_VEL
LIN {X 0,Y 504.71,Z 1041.225,A -85,B 0,C 180,E1 23682.82,E2 23682.82} C_VEL
LIN {X 0,Y 504.343,Z 1050.99,A -85,B 0,C 180,E1 23680.856,E2 23680.856} C_VEL
LIN {X 0,Y 504.102,Z 1059.175,A -85,B 0,C 180,E1 23678.785,E2 23678.785} C_VEL
LIN {X 0,Y 503.982,Z 1065.411,A -85,B 0,C 180,E1 23676.722,E2 23676.722} C_VEL
LIN {X 0,Y 503.929,Z 1069.876,A -85,B 0,C 180,E1 23674.666,E2 23674.666} C_VEL
LIN {X 0,Y 503.911,Z 1072.792,A -85,B 0,C 180,E1 23672.502,E2 23672.502} C_VEL
LIN {X 0,Y 503.908,Z 1073.939,A -85,B 0,C 180,E1 23670.341,E2 23670.341} C_VEL
LIN {X 0,Y 503.912,Z 1073.413,A -85,B 0,C 180,E1 23668.295,E2 23668.295} C_VEL
LIN {X 0,Y 503.92,Z 1071.159,A -85,B 0,C 180,E1 23666.132,E2 23666.132} C_VEL
LIN {X 0,Y 503.95,Z 1067.351,A -85,B 0,C 180,E1 23664.078,E2 23664.078} C_VEL
LIN {X 0,Y 504.041,Z 1061.821,A -85,B 0,C 180,E1 23662.018,E2 23662.018} C_VEL
LIN {X 0,Y 504.234,Z 1054.426,A -85,B 0,C 180,E1 23659.951,E2 23659.951} C_VEL
LIN {X 0,Y 504.538,Z 1045.517,A -85,B 0,C 180,E1 23657.99,E2 23657.99} C_VEL
LIN {X 0,Y 504.977,Z 1035.151,A -85,B 0,C 180,E1 23656.138,E2 23656.138} C_VEL
LIN {X 0,Y 505.557,Z 1023.351,A -85,B 0,C 180,E1 23654.397,E2 23654.397} C_VEL
LIN {X 0,Y 506.264,Z 1010.069,A -85,B 0,C 180,E1 23652.768,E2 23652.768} C_VEL
LIN {X 0,Y 506.947,Z 996.653,A -85,B 0,C 180,E1 23651.426,E2 23651.426} C_VEL
LIN {X 0,Y 507.695,Z 981.092,A -85,B 0,C 180,E1 23650.14,E2 23650.14} C_VEL
LIN {X 0,Y 508.429,Z 964.771,A -85,B 0,C 180,E1 23649.028,E2 23649.028} C_VEL
LIN {X 0,Y 509.188,Z 947.117,A -85,B 0,C 180,E1 23648.059,E2 23648.059} C_VEL
LIN {X 0,Y 509.8,Z 929.548,A -85,B 0,C 180,E1 23647.308,E2 23647.308} C_VEL
LIN {X 0,Y 510.354,Z 910.911,A -85,B 0,C 180,E1 23646.725,E2 23646.725} C_VEL
LIN {X 0,Y 510.721,Z 891.627,A -85,B 0,C 180,E1 23646.335,E2 23646.335} C_VEL
LIN {X 0,Y 511.897,Z 704.171,A -85,B 0,C 180,E1 23643.659,E2 23643.659} C_VEL
LIN {X 0,Y 510.161,Z 692.019,A -85,B 0,C 180,E1 23643.389,E2 23643.389} C_VEL
LIN {X 0,Y 511.715,Z 649.142,A -85,B 0,C 180,E1 23640.051,E2 23640.051} C_VEL
LIN {X 0,Y 513.037,Z 617.094,A -85,B 0,C 180,E1 23637.489,E2 23637.489} C_VEL
LIN {X 0,Y 505.669,Z 596.016,A -85,B 0,C 180,E1 23635.143,E2 23635.143} C_VEL
LIN {X 0,Y 504.716,Z 593.125,A -85,B 0,C 180,E1 23634.751,E2 23634.751} C_VEL
LIN {X 0,Y 504.649,Z 592.936,A -85,B 0,C 180,E1 23631.318,E2 23631.318} C_VEL
LIN {X 0,Y 504.707,Z 592.93,A -85,B 0,C 180,E1 23627.964,E2 23627.964} C_VEL
LIN {X 0,Y 504.671,Z 592.931,A -85,B 0,C 180,E1 23624.535,E2 23624.535} C_VEL
LIN {X 0,Y 504.657,Z 592.934,A -85,B 0,C 180,E1 23621.131,E2 23621.131} C_VEL
LIN {X 0,Y 504.715,Z 592.923,A -85,B 0,C 180,E1 23617.744,E2 23617.744} C_VEL
LIN {X 0,Y 504.656,Z 592.93,A -85,B 0,C 180,E1 23614.379,E2 23614.379} C_VEL
LIN {X 0,Y 504.664,Z 592.934,A -85,B 0,C 180,E1 23610.873,E2 23610.873} C_VEL
LIN {X 0,Y 504.71,Z 592.921,A -85,B 0,C 180,E1 23607.489,E2 23607.489} C_VEL
LIN {X 0,Y 504.655,Z 592.926,A -85,B 0,C 180,E1 23604.088,E2 23604.088} C_VEL
LIN {X 0,Y 504.683,Z 592.931,A -85,B 0,C 180,E1 23600.649,E2 23600.649} C_VEL
LIN {X 0,Y 504.695,Z 592.926,A -85,B 0,C 180,E1 23597.273,E2 23597.273} C_VEL
LIN {X 0,Y 504.656,Z 592.927,A -85,B 0,C 180,E1 23593.871,E2 23593.871} C_VEL
LIN {X 0,Y 504.707,Z 592.926,A -85,B 0,C 180,E1 23590.501,E2 23590.501} C_VEL
LIN {X 0,Y 504.685,Z 592.928,A -85,B 0,C 180,E1 23586.994,E2 23586.994} C_VEL
LIN {X 0,Y 504.662,Z 592.93,A -85,B 0,C 180,E1 23583.521,E2 23583.521} C_VEL
LIN {X 0,Y 504.713,Z 592.922,A -85,B 0,C 180,E1 23580.113,E2 23580.113} C_VEL
LIN {X 0,Y 504.686,Z 592.927,A -85,B 0,C 180,E1 23576.592,E2 23576.592} C_VEL
LIN {X 0,Y 504.666,Z 592.931,A -85,B 0,C 180,E1 23573.058,E2 23573.058} C_VEL
LIN {X 0,Y 504.707,Z 592.925,A -85,B 0,C 180,E1 23569.614,E2 23569.614} C_VEL
LIN {X 0,Y 504.694,Z 592.92,A -85,B 0,C 180,E1 23566.108,E2 23566.108} C_VEL
LIN {X 0,Y 504.67,Z 592.926,A -85,B 0,C 180,E1 23562.592,E2 23562.592} C_VEL
LIN {X 0,Y 504.71,Z 592.925,A -85,B 0,C 180,E1 23559.109,E2 23559.109} C_VEL
LIN {X 0,Y 504.705,Z 592.922,A -85,B 0,C 180,E1 23555.54,E2 23555.54} C_VEL
LIN {X 0,Y 504.674,Z 592.931,A -85,B 0,C 180,E1 23552.082,E2 23552.082} C_VEL
LIN {X 0,Y 504.707,Z 592.928,A -85,B 0,C 180,E1 23548.599,E2 23548.599} C_VEL
LIN {X 0,Y 504.706,Z 592.931,A -85,B 0,C 180,E1 23545.073,E2 23545.073} C_VEL
LIN {X 0,Y 504.68,Z 592.933,A -85,B 0,C 180,E1 23541.531,E2 23541.531} C_VEL
LIN {X 0,Y 504.745,Z 593.195,A -85,B 0,C 180,E1 23541.024,E2 23541.024} C_VEL
LIN {X 0,Y 509.606,Z 610.677,A -85,B 0,C 180,E1 23538.308,E2 23538.308} C_VEL
LIN {X 0,Y 509.862,Z 613.789,A -85,B 0,C 180,E1 23537.88,E2 23537.88} C_VEL
LIN {X 0,Y 508.509,Z 642.304,A -85,B 0,C 180,E1 23534.268,E2 23534.268} C_VEL
LIN {X 0,Y 508.345,Z 646.04,A -85,B 0,C 180,E1 23533.799,E2 23533.799} C_VEL
LIN {X 0,Y 507.176,Z 651.414,A -85,B 0,C 180,E1 23533.181,E2 23533.181} C_VEL
LIN {X 0,Y 500.383,Z 667.203,A -85,B 0,C 180,E1 23531.548,E2 23531.548} C_VEL
LIN {X 0,Y 499.724,Z 671.053,A -85,B 0,C 180,E1 23531.093,E2 23531.093} C_VEL
LIN {X 0,Y 498.58,Z 701.178,A -85,B 0,C 180,E1 23527.347,E2 23527.347} C_VEL
LIN {X 0,Y 498.366,Z 709.237,A -85,B 0,C 180,E1 23526.387,E2 23526.387} C_VEL
LIN {X 0,Y 500.324,Z 721.79,A -85,B 0,C 180,E1 23526.085,E2 23526.085} C_VEL
LIN {X 0,Y 499.43,Z 823.926,A -85,B 0,C 180,E1 23524.524,E2 23524.524} C_VEL
LIN {X 0,Y 499.176,Z 838.926,A -85,B 0,C 180,E1 23524.081,E2 23524.081} C_VEL
LIN {X 0,Y 498.77,Z 853.606,A -85,B 0,C 180,E1 23523.409,E2 23523.409} C_VEL
LIN {X 0,Y 498.295,Z 866.961,A -85,B 0,C 180,E1 23522.567,E2 23522.567} C_VEL
LIN {X 0,Y 497.806,Z 879.328,A -85,B 0,C 180,E1 23521.549,E2 23521.549} C_VEL
LIN {X 0,Y 497.338,Z 890.964,A -85,B 0,C 180,E1 23520.306,E2 23520.306} C_VEL
LIN {X 0,Y 496.917,Z 900.517,A -85,B 0,C 180,E1 23519.007,E2 23519.007} C_VEL
LIN {X 0,Y 496.583,Z 908.744,A -85,B 0,C 180,E1 23517.587,E2 23517.587} C_VEL
LIN {X 0,Y 496.345,Z 915.536,A -85,B 0,C 180,E1 23516.045,E2 23516.045} C_VEL
LIN {X 0,Y 496.198,Z 920.877,A -85,B 0,C 180,E1 23514.383,E2 23514.383} C_VEL
LIN {X 0,Y 496.129,Z 924.54,A -85,B 0,C 180,E1 23512.628,E2 23512.628} C_VEL
LIN {X 0,Y 496.103,Z 926.298,A -85,B 0,C 180,E1 23510.899,E2 23510.899} C_VEL
LIN {X 0,Y 496.097,Z 926.373,A -85,B 0,C 180,E1 23509.179,E2 23509.179} C_VEL
LIN {X 0,Y 496.118,Z 924.588,A -85,B 0,C 180,E1 23507.354,E2 23507.354} C_VEL
LIN {X 0,Y 496.18,Z 920.917,A -85,B 0,C 180,E1 23505.585,E2 23505.585} C_VEL
LIN {X 0,Y 496.31,Z 915.863,A -85,B 0,C 180,E1 23503.99,E2 23503.99} C_VEL
LIN {X 0,Y 496.549,Z 908.546,A -85,B 0,C 180,E1 23502.324,E2 23502.324} C_VEL
LIN {X 0,Y 496.908,Z 899.489,A -85,B 0,C 180,E1 23500.785,E2 23500.785} C_VEL
LIN {X 0,Y 497.322,Z 889.648,A -85,B 0,C 180,E1 23499.489,E2 23499.489} C_VEL
LIN {X 0,Y 497.754,Z 878.406,A -85,B 0,C 180,E1 23498.316,E2 23498.316} C_VEL
LIN {X 0,Y 498.278,Z 865.318,A -85,B 0,C 180,E1 23497.262,E2 23497.262} C_VEL
LIN {X 0,Y 498.725,Z 851.858,A -85,B 0,C 180,E1 23496.446,E2 23496.446} C_VEL
LIN {X 0,Y 499.098,Z 837.562,A -85,B 0,C 180,E1 23495.817,E2 23495.817} C_VEL
LIN {X 0,Y 499.361,Z 821.857,A -85,B 0,C 180,E1 23495.375,E2 23495.375} C_VEL
LIN {X 0,Y 499.961,Z 719.58,A -85,B 0,C 180,E1 23493.833,E2 23493.833} C_VEL
LIN {X 0,Y 498.249,Z 709.023,A -85,B 0,C 180,E1 23493.566,E2 23493.566} C_VEL
LIN {X 0,Y 499.233,Z 679.891,A -85,B 0,C 180,E1 23490,E2 23490} C_VEL
LIN {X 0,Y 500.471,Z 650.635,A -85,B 0,C 180,E1 23486.334,E2 23486.334} C_VEL
LIN {X 0,Y 501.848,Z 621.845,A -85,B 0,C 180,E1 23482.674,E2 23482.674} C_VEL
LIN {X 0,Y 502.202,Z 613.848,A -85,B 0,C 180,E1 23481.643,E2 23481.643} C_VEL
LIN {X 0,Y 497.172,Z 595.65,A -85,B 0,C 180,E1 23478.868,E2 23478.868} C_VEL
LIN {X 0,Y 496.78,Z 594.013,A -85,B 0,C 180,E1 23478.574,E2 23478.574} C_VEL
LIN {X 0,Y 496.759,Z 593.918,A -85,B 0,C 180,E1 23474.951,E2 23474.951} C_VEL
LIN {X 0,Y 496.757,Z 593.919,A -85,B 0,C 180,E1 23471.446,E2 23471.446} C_VEL
LIN {X 0,Y 496.753,Z 593.916,A -85,B 0,C 180,E1 23467.803,E2 23467.803} C_VEL
LIN {X 0,Y 496.764,Z 593.914,A -85,B 0,C 180,E1 23464.23,E2 23464.23} C_VEL
LIN {X 0,Y 496.769,Z 593.9,A -85,B 0,C 180,E1 23460.586,E2 23460.586} C_VEL
LIN {X 0,Y 496.746,Z 593.906,A -85,B 0,C 180,E1 23457.072,E2 23457.072} C_VEL
LIN {X 0,Y 496.764,Z 593.912,A -85,B 0,C 180,E1 23453.575,E2 23453.575} C_VEL
LIN {X 0,Y 496.769,Z 593.92,A -85,B 0,C 180,E1 23450.054,E2 23450.054} C_VEL
LIN {X 0,Y 496.745,Z 593.909,A -85,B 0,C 180,E1 23446.497,E2 23446.497} C_VEL
LIN {X 0,Y 496.75,Z 593.914,A -85,B 0,C 180,E1 23442.87,E2 23442.87} C_VEL
LIN {X 0,Y 496.767,Z 593.914,A -85,B 0,C 180,E1 23439.385,E2 23439.385} C_VEL
LIN {X 0,Y 496.752,Z 593.92,A -85,B 0,C 180,E1 23435.855,E2 23435.855} C_VEL
LIN {X 0,Y 496.739,Z 593.91,A -85,B 0,C 180,E1 23432.285,E2 23432.285} C_VEL
LIN {X 0,Y 496.77,Z 593.913,A -85,B 0,C 180,E1 23428.885,E2 23428.885} C_VEL
LIN {X 0,Y 496.752,Z 593.904,A -85,B 0,C 180,E1 23425.344,E2 23425.344} C_VEL
LIN {X 0,Y 496.735,Z 593.917,A -85,B 0,C 180,E1 23421.863,E2 23421.863} C_VEL
LIN {X 0,Y 496.769,Z 593.899,A -85,B 0,C 180,E1 23418.421,E2 23418.421} C_VEL
LIN {X 0,Y 496.749,Z 593.915,A -85,B 0,C 180,E1 23414.93,E2 23414.93} C_VEL
LIN {X 0,Y 496.731,Z 593.915,A -85,B 0,C 180,E1 23411.377,E2 23411.377} C_VEL
LIN {X 0,Y 496.771,Z 593.904,A -85,B 0,C 180,E1 23407.867,E2 23407.867} C_VEL
LIN {X 0,Y 496.755,Z 593.922,A -85,B 0,C 180,E1 23404.387,E2 23404.387} C_VEL
LIN {X 0,Y 496.724,Z 593.905,A -85,B 0,C 180,E1 23400.923,E2 23400.923} C_VEL
LIN {X 0,Y 496.767,Z 593.914,A -85,B 0,C 180,E1 23397.462,E2 23397.462} C_VEL
LIN {X 0,Y 496.764,Z 593.908,A -85,B 0,C 180,E1 23393.882,E2 23393.882} C_VEL
LIN {X 0,Y 496.723,Z 593.916,A -85,B 0,C 180,E1 23390.5,E2 23390.5} C_VEL
LIN {X 0,Y 496.77,Z 593.908,A -85,B 0,C 180,E1 23387.091,E2 23387.091} C_VEL
LIN {X 0,Y 496.744,Z 593.917,A -85,B 0,C 180,E1 23383.633,E2 23383.633} C_VEL
LIN {X 0,Y 496.721,Z 593.915,A -85,B 0,C 180,E1 23380.112,E2 23380.112} C_VEL
LIN {X 0,Y 496.775,Z 593.916,A -85,B 0,C 180,E1 23376.766,E2 23376.766} C_VEL
LIN {X 0,Y 496.732,Z 593.913,A -85,B 0,C 180,E1 23373.329,E2 23373.329} C_VEL
LIN {X 0,Y 496.727,Z 593.915,A -85,B 0,C 180,E1 23369.92,E2 23369.92} C_VEL
LIN {X 0,Y 496.775,Z 593.916,A -85,B 0,C 180,E1 23366.532,E2 23366.532} C_VEL
LIN {X 0,Y 496.717,Z 593.923,A -85,B 0,C 180,E1 23363.141,E2 23363.141} C_VEL
LIN {X 0,Y 496.732,Z 593.92,A -85,B 0,C 180,E1 23359.598,E2 23359.598} C_VEL
LIN {X 0,Y 496.775,Z 593.915,A -85,B 0,C 180,E1 23356.1,E2 23356.1} C_VEL
LIN {X 0,Y 496.716,Z 593.92,A -85,B 0,C 180,E1 23352.716,E2 23352.716} C_VEL
LIN {X 0,Y 496.728,Z 593.92,A -85,B 0,C 180,E1 23349.198,E2 23349.198} C_VEL
LIN {X 0,Y 496.78,Z 594.003,A -85,B 0,C 180,E1 23345.796,E2 23345.796} C_VEL
LIN {X 0,Y 496.905,Z 594.663,A -85,B 0,C 180,E1 23345.618,E2 23345.618} C_VEL
LIN {X 0,Y 505.176,Z 618.196,A -85,B 0,C 180,E1 23342.945,E2 23342.945} C_VEL
LIN {X 0,Y 505.819,Z 621.02,A -85,B 0,C 180,E1 23342.66,E2 23342.66} C_VEL
LIN {X 0,Y 503.763,Z 665.146,A -85,B 0,C 180,E1 23339.096,E2 23339.096} C_VEL
LIN {X 0,Y 502.67,Z 692.368,A -85,B 0,C 180,E1 23336.954,E2 23336.954} C_VEL
LIN {X 0,Y 504.637,Z 707.976,A -85,B 0,C 180,E1 23336.622,E2 23336.622} C_VEL
LIN {X 0,Y 503.045,Z 899.75,A -85,B 0,C 180,E1 23333.824,E2 23333.824} C_VEL
LIN {X 0,Y 502.516,Z 918.876,A -85,B 0,C 180,E1 23333.335,E2 23333.335} C_VEL
LIN {X 0,Y 501.865,Z 937.441,A -85,B 0,C 180,E1 23332.645,E2 23332.645} C_VEL
LIN {X 0,Y 501.145,Z 954.903,A -85,B 0,C 180,E1 23331.784,E2 23331.784} C_VEL
LIN {X 0,Y 500.298,Z 972.055,A -85,B 0,C 180,E1 23330.717,E2 23330.717} C_VEL
LIN {X 0,Y 499.483,Z 988.371,A -85,B 0,C 180,E1 23329.466,E2 23329.466} C_VEL
LIN {X 0,Y 498.646,Z 1004.254,A -85,B 0,C 180,E1 23327.987,E2 23327.987} C_VEL
LIN {X 0,Y 497.921,Z 1018.01,A -85,B 0,C 180,E1 23326.448,E2 23326.448} C_VEL
LIN {X 0,Y 497.268,Z 1031.218,A -85,B 0,C 180,E1 23324.676,E2 23324.676} C_VEL
LIN {X 0,Y 496.804,Z 1041.224,A -85,B 0,C 180,E1 23323.027,E2 23323.027} C_VEL
LIN {X 0,Y 496.398,Z 1050.99,A -85,B 0,C 180,E1 23321.032,E2 23321.032} C_VEL
LIN {X 0,Y 496.123,Z 1059.174,A -85,B 0,C 180,E1 23318.928,E2 23318.928} C_VEL
LIN {X 0,Y 495.991,Z 1065.411,A -85,B 0,C 180,E1 23316.831,E2 23316.831} C_VEL
LIN {X 0,Y 495.929,Z 1069.875,A -85,B 0,C 180,E1 23314.742,E2 23314.742} C_VEL
LIN {X 0,Y 495.911,Z 1072.792,A -85,B 0,C 180,E1 23312.543,E2 23312.543} C_VEL
LIN {X 0,Y 495.908,Z 1073.939,A -85,B 0,C 180,E1 23310.347,E2 23310.347} C_VEL
LIN {X 0,Y 495.912,Z 1073.413,A -85,B 0,C 180,E1 23308.267,E2 23308.267} C_VEL
LIN {X 0,Y 495.921,Z 1071.159,A -85,B 0,C 180,E1 23306.07,E2 23306.07} C_VEL
LIN {X 0,Y 495.956,Z 1067.35,A -85,B 0,C 180,E1 23303.983,E2 23303.983} C_VEL
LIN {X 0,Y 496.057,Z 1061.821,A -85,B 0,C 180,E1 23301.889,E2 23301.889} C_VEL
LIN {X 0,Y 496.271,Z 1054.426,A -85,B 0,C 180,E1 23299.788,E2 23299.788} C_VEL
LIN {X 0,Y 496.612,Z 1045.516,A -85,B 0,C 180,E1 23297.796,E2 23297.796} C_VEL
LIN {X 0,Y 497.054,Z 1035.78,A -85,B 0,C 180,E1 23296.032,E2 23296.032} C_VEL
LIN {X 0,Y 497.59,Z 1024.479,A -85,B 0,C 180,E1 23294.38,E2 23294.38} C_VEL
LIN {X 0,Y 498.291,Z 1010.866,A -85,B 0,C 180,E1 23292.724,E2 23292.724} C_VEL
LIN {X 0,Y 499.089,Z 995.643,A -85,B 0,C 180,E1 23291.183,E2 23291.183} C_VEL
LIN {X 0,Y 499.92,Z 979.437,A -85,B 0,C 180,E1 23289.828,E2 23289.828} C_VEL
LIN {X 0,Y 500.736,Z 962.811,A -85,B 0,C 180,E1 23288.69,E2 23288.69} C_VEL
LIN {X 0,Y 501.522,Z 945.557,A -85,B 0,C 180,E1 23287.741,E2 23287.741} C_VEL
LIN {X 0,Y 502.192,Z 927.475,A -85,B 0,C 180,E1 23286.969,E2 23286.969} C_VEL
LIN {X 0,Y 502.789,Z 908.397,A -85,B 0,C 180,E1 23286.382,E2 23286.382} C_VEL
LIN {X 0,Y 503.165,Z 888.373,A -85,B 0,C 180,E1 23285.998,E2 23285.998} C_VEL
LIN {X 0,Y 504.406,Z 705.088,A -85,B 0,C 180,E1 23283.348,E2 23283.348} C_VEL
LIN {X 0,Y 502.612,Z 692.231,A -85,B 0,C 180,E1 23283.059,E2 23283.059} C_VEL
LIN {X 0,Y 504.337,Z 648.9,A -85,B 0,C 180,E1 23279.633,E2 23279.633} C_VEL
LIN {X 0,Y 505.752,Z 619.966,A -85,B 0,C 180,E1 23277.262,E2 23277.262} C_VEL
LIN {X 0,Y 498.798,Z 599.917,A -85,B 0,C 180,E1 23274.98,E2 23274.98} C_VEL
LIN {X 0,Y 496.798,Z 594.121,A -85,B 0,C 180,E1 23274.233,E2 23274.233} C_VEL
LIN {X 0,Y 496.716,Z 593.922,A -85,B 0,C 180,E1 23270.946,E2 23270.946} C_VEL
LIN {X 0,Y 496.724,Z 593.923,A -85,B 0,C 180,E1 23267.442,E2 23267.442} C_VEL
LIN {X 0,Y 496.773,Z 593.915,A -85,B 0,C 180,E1 23263.978,E2 23263.978} C_VEL
LIN {X 0,Y 496.719,Z 593.921,A -85,B 0,C 180,E1 23260.555,E2 23260.555} C_VEL
LIN {X 0,Y 496.717,Z 593.923,A -85,B 0,C 180,E1 23256.952,E2 23256.952} C_VEL
LIN {X 0,Y 496.774,Z 593.917,A -85,B 0,C 180,E1 23253.565,E2 23253.565} C_VEL
LIN {X 0,Y 496.718,Z 593.92,A -85,B 0,C 180,E1 23250.214,E2 23250.214} C_VEL
LIN {X 0,Y 496.725,Z 593.923,A -85,B 0,C 180,E1 23246.654,E2 23246.654} C_VEL
LIN {X 0,Y 496.773,Z 593.909,A -85,B 0,C 180,E1 23243.234,E2 23243.234} C_VEL
LIN {X 0,Y 496.72,Z 593.915,A -85,B 0,C 180,E1 23239.888,E2 23239.888} C_VEL
LIN {X 0,Y 496.735,Z 593.921,A -85,B 0,C 180,E1 23236.367,E2 23236.367} C_VEL
LIN {X 0,Y 496.77,Z 593.912,A -85,B 0,C 180,E1 23232.909,E2 23232.909} C_VEL
LIN {X 0,Y 496.724,Z 593.908,A -85,B 0,C 180,E1 23229.486,E2 23229.486} C_VEL
LIN {X 0,Y 496.742,Z 593.917,A -85,B 0,C 180,E1 23226.008,E2 23226.008} C_VEL
LIN {X 0,Y 496.766,Z 593.915,A -85,B 0,C 180,E1 23222.538,E2 23222.538} C_VEL
LIN {X 0,Y 496.726,Z 593.914,A -85,B 0,C 180,E1 23219.077,E2 23219.077} C_VEL
LIN {X 0,Y 496.742,Z 593.912,A -85,B 0,C 180,E1 23215.497,E2 23215.497} C_VEL
LIN {X 0,Y 496.774,Z 593.918,A -85,B 0,C 180,E1 23211.994,E2 23211.994} C_VEL
LIN {X 0,Y 496.736,Z 593.918,A -85,B 0,C 180,E1 23208.505,E2 23208.505} C_VEL
LIN {X 0,Y 496.737,Z 593.922,A -85,B 0,C 180,E1 23204.95,E2 23204.95} C_VEL
LIN {X 0,Y 496.771,Z 593.916,A -85,B 0,C 180,E1 23201.44,E2 23201.44} C_VEL
LIN {X 0,Y 496.749,Z 593.917,A -85,B 0,C 180,E1 23197.889,E2 23197.889} C_VEL
LIN {X 0,Y 496.738,Z 593.92,A -85,B 0,C 180,E1 23194.357,E2 23194.357} C_VEL
LIN {X 0,Y 496.774,Z 593.916,A -85,B 0,C 180,E1 23190.851,E2 23190.851} C_VEL
LIN {X 0,Y 496.766,Z 593.918,A -85,B 0,C 180,E1 23187.28,E2 23187.28} C_VEL
LIN {X 0,Y 496.74,Z 593.923,A -85,B 0,C 180,E1 23183.716,E2 23183.716} C_VEL
LIN {X 0,Y 496.777,Z 594.171,A -85,B 0,C 180,E1 23181.53,E2 23181.53} C_VEL
LIN {X 0,Y 501.65,Z 611.224,A -85,B 0,C 180,E1 23178.796,E2 23178.796} C_VEL
LIN {X 0,Y 502.456,Z 615.291,A -85,B 0,C 180,E1 23178.192,E2 23178.192} C_VEL
LIN {X 0,Y 500.994,Z 643.561,A -85,B 0,C 180,E1 23174.562,E2 23174.562} C_VEL
LIN {X 0,Y 499.724,Z 671.053,A -85,B 0,C 180,E1 23171.093,E2 23171.093} C_VEL
LIN {X 0,Y 498.578,Z 676.458,A -85,B 0,C 180,E1 23170.467,E2 23170.467} C_VEL
LIN {X 0,Y 491.803,Z 692.243,A -85,B 0,C 180,E1 23168.806,E2 23168.806} C_VEL
LIN {X 0,Y 491.131,Z 696.112,A -85,B 0,C 180,E1 23168.346,E2 23168.346} C_VEL
LIN {X 0,Y 490.704,Z 709.267,A -85,B 0,C 180,E1 23166.746,E2 23166.746} C_VEL
LIN {X 0,Y 492.889,Z 722.73,A -85,B 0,C 180,E1 23166.416,E2 23166.416} C_VEL
LIN {X 0,Y 491.9,Z 824.664,A -85,B 0,C 180,E1 23164.827,E2 23164.827} C_VEL
LIN {X 0,Y 491.631,Z 839.53,A -85,B 0,C 180,E1 23164.38,E2 23164.38} C_VEL
LIN {X 0,Y 491.212,Z 853.782,A -85,B 0,C 180,E1 23163.724,E2 23163.724} C_VEL
LIN {X 0,Y 490.712,Z 867.074,A -85,B 0,C 180,E1 23162.889,E2 23162.889} C_VEL
LIN {X 0,Y 490.152,Z 880.021,A -85,B 0,C 180,E1 23161.817,E2 23161.817} C_VEL
LIN {X 0,Y 489.632,Z 891.666,A -85,B 0,C 180,E1 23160.562,E2 23160.562} C_VEL
LIN {X 0,Y 489.154,Z 901.507,A -85,B 0,C 180,E1 23159.212,E2 23159.212} C_VEL
LIN {X 0,Y 488.754,Z 910.259,A -85,B 0,C 180,E1 23157.67,E2 23157.67} C_VEL
LIN {X 0,Y 488.471,Z 917.427,A -85,B 0,C 180,E1 23155.979,E2 23155.979} C_VEL
LIN {X 0,Y 488.307,Z 922.489,A -85,B 0,C 180,E1 23154.303,E2 23154.303} C_VEL
LIN {X 0,Y 488.223,Z 925.969,A -85,B 0,C 180,E1 23152.518,E2 23152.518} C_VEL
LIN {X 0,Y 488.193,Z 927.65,A -85,B 0,C 180,E1 23150.613,E2 23150.613} C_VEL
LIN {X 0,Y 488.191,Z 927.326,A -85,B 0,C 180,E1 23148.757,E2 23148.757} C_VEL
LIN {X 0,Y 488.223,Z 925.23,A -85,B 0,C 180,E1 23146.981,E2 23146.981} C_VEL
LIN {X 0,Y 488.317,Z 921.267,A -85,B 0,C 180,E1 23145.194,E2 23145.194} C_VEL
LIN {X 0,Y 488.496,Z 915.559,A -85,B 0,C 180,E1 23143.493,E2 23143.493} C_VEL
LIN {X 0,Y 488.771,Z 908.339,A -85,B 0,C 180,E1 23141.924,E2 23141.924} C_VEL
LIN {X 0,Y 489.166,Z 899.739,A -85,B 0,C 180,E1 23140.481,E2 23140.481} C_VEL
LIN {X 0,Y 489.673,Z 888.678,A -85,B 0,C 180,E1 23139.046,E2 23139.046} C_VEL
LIN {X 0,Y 490.167,Z 876.824,A -85,B 0,C 180,E1 23137.855,E2 23137.855} C_VEL
LIN {X 0,Y 490.694,Z 864.708,A -85,B 0,C 180,E1 23136.905,E2 23136.905} C_VEL
LIN {X 0,Y 491.183,Z 850.809,A -85,B 0,C 180,E1 23136.076,E2 23136.076} C_VEL
LIN {X 0,Y 491.57,Z 836.112,A -85,B 0,C 180,E1 23135.456,E2 23135.456} C_VEL
LIN {X 0,Y 491.81,Z 821.325,A -85,B 0,C 180,E1 23135.057,E2 23135.057} C_VEL
LIN {X 0,Y 492.487,Z 720.485,A -85,B 0,C 180,E1 23133.514,E2 23133.514} C_VEL
LIN {X 0,Y 490.549,Z 708.88,A -85,B 0,C 180,E1 23133.213,E2 23133.213} C_VEL
LIN {X 0,Y 491.648,Z 679.281,A -85,B 0,C 180,E1 23129.534,E2 23129.534} C_VEL
LIN {X 0,Y 492.944,Z 650.82,A -85,B 0,C 180,E1 23125.929,E2 23125.929} C_VEL
LIN {X 0,Y 494.44,Z 621.99,A -85,B 0,C 180,E1 23122.213,E2 23122.213} C_VEL
LIN {X 0,Y 494.521,Z 615.672,A -85,B 0,C 180,E1 23121.379,E2 23121.379} C_VEL
LIN {X 0,Y 489.431,Z 597.149,A -85,B 0,C 180,E1 23118.511,E2 23118.511} C_VEL
LIN {X 0,Y 488.832,Z 595.035,A -85,B 0,C 180,E1 23118.137,E2 23118.137} C_VEL
LIN {X 0,Y 488.826,Z 594.904,A -85,B 0,C 180,E1 23114.579,E2 23114.579} C_VEL
LIN {X 0,Y 488.824,Z 594.907,A -85,B 0,C 180,E1 23110.909,E2 23110.909} C_VEL
LIN {X 0,Y 488.813,Z 594.898,A -85,B 0,C 180,E1 23107.384,E2 23107.384} C_VEL
LIN {X 0,Y 488.82,Z 594.903,A -85,B 0,C 180,E1 23103.78,E2 23103.78} C_VEL
LIN {X 0,Y 488.823,Z 594.883,A -85,B 0,C 180,E1 23100.195,E2 23100.195} C_VEL
LIN {X 0,Y 488.825,Z 594.899,A -85,B 0,C 180,E1 23096.568,E2 23096.568} C_VEL
LIN {X 0,Y 488.805,Z 594.904,A -85,B 0,C 180,E1 23093.031,E2 23093.031} C_VEL
LIN {X 0,Y 488.832,Z 594.903,A -85,B 0,C 180,E1 23089.543,E2 23089.543} C_VEL
LIN {X 0,Y 488.83,Z 594.903,A -85,B 0,C 180,E1 23085.885,E2 23085.885} C_VEL
LIN {X 0,Y 488.807,Z 594.907,A -85,B 0,C 180,E1 23082.297,E2 23082.297} C_VEL
LIN {X 0,Y 488.806,Z 594.903,A -85,B 0,C 180,E1 23078.612,E2 23078.612} C_VEL
LIN {X 0,Y 488.827,Z 594.894,A -85,B 0,C 180,E1 23075.084,E2 23075.084} C_VEL
LIN {X 0,Y 488.824,Z 594.905,A -85,B 0,C 180,E1 23071.465,E2 23071.465} C_VEL
LIN {X 0,Y 488.798,Z 594.905,A -85,B 0,C 180,E1 23067.91,E2 23067.91} C_VEL
LIN {X 0,Y 488.823,Z 594.897,A -85,B 0,C 180,E1 23064.405,E2 23064.405} C_VEL
LIN {X 0,Y 488.833,Z 594.904,A -85,B 0,C 180,E1 23060.811,E2 23060.811} C_VEL
LIN {X 0,Y 488.795,Z 594.891,A -85,B 0,C 180,E1 23057.254,E2 23057.254} C_VEL
LIN {X 0,Y 488.799,Z 594.905,A -85,B 0,C 180,E1 23053.606,E2 23053.606} C_VEL
LIN {X 0,Y 488.831,Z 594.889,A -85,B 0,C 180,E1 23050.132,E2 23050.132} C_VEL
LIN {X 0,Y 488.805,Z 594.902,A -85,B 0,C 180,E1 23046.578,E2 23046.578} C_VEL
LIN {X 0,Y 488.791,Z 594.904,A -85,B 0,C 180,E1 23043.049,E2 23043.049} C_VEL
LIN {X 0,Y 488.831,Z 594.895,A -85,B 0,C 180,E1 23039.531,E2 23039.531} C_VEL
LIN {X 0,Y 488.819,Z 594.911,A -85,B 0,C 180,E1 23036.012,E2 23036.012} C_VEL
LIN {X 0,Y 488.783,Z 594.892,A -85,B 0,C 180,E1 23032.596,E2 23032.596} C_VEL
LIN {X 0,Y 488.827,Z 594.904,A -85,B 0,C 180,E1 23029.154,E2 23029.154} C_VEL
LIN {X 0,Y 488.809,Z 594.898,A -85,B 0,C 180,E1 23025.67,E2 23025.67} C_VEL
LIN {X 0,Y 488.784,Z 594.908,A -85,B 0,C 180,E1 23022.254,E2 23022.254} C_VEL
LIN {X 0,Y 488.835,Z 594.899,A -85,B 0,C 180,E1 23018.775,E2 23018.775} C_VEL
LIN {X 0,Y 488.808,Z 594.909,A -85,B 0,C 180,E1 23015.26,E2 23015.26} C_VEL
LIN {X 0,Y 488.779,Z 594.909,A -85,B 0,C 180,E1 23011.801,E2 23011.801} C_VEL
LIN {X 0,Y 488.835,Z 594.904,A -85,B 0,C 180,E1 23008.425,E2 23008.425} C_VEL
LIN {X 0,Y 488.801,Z 594.906,A -85,B 0,C 180,E1 23004.907,E2 23004.907} C_VEL
LIN {X 0,Y 488.772,Z 594.906,A -85,B 0,C 180,E1 23001.393,E2 23001.393} C_VEL
LIN {X 0,Y 488.833,Z 594.904,A -85,B 0,C 180,E1 22998.022,E2 22998.022} C_VEL
LIN {X 0,Y 488.793,Z 594.91,A -85,B 0,C 180,E1 22994.558,E2 22994.558} C_VEL
LIN {X 0,Y 488.775,Z 594.911,A -85,B 0,C 180,E1 22991.046,E2 22991.046} C_VEL
LIN {X 0,Y 488.836,Z 594.908,A -85,B 0,C 180,E1 22987.668,E2 22987.668} C_VEL
LIN {X 0,Y 488.836,Z 595.191,A -85,B 0,C 180,E1 22986.197,E2 22986.197} C_VEL
LIN {X 0,Y 496.721,Z 617.662,A -85,B 0,C 180,E1 22983.556,E2 22983.556} C_VEL
LIN {X 0,Y 498.504,Z 623.438,A -85,B 0,C 180,E1 22982.926,E2 22982.926} C_VEL
LIN {X 0,Y 496.238,Z 667.28,A -85,B 0,C 180,E1 22979.316,E2 22979.316} C_VEL
LIN {X 0,Y 495.151,Z 692.565,A -85,B 0,C 180,E1 22977.299,E2 22977.299} C_VEL
LIN {X 0,Y 497.19,Z 708.905,A -85,B 0,C 180,E1 22976.946,E2 22976.946} C_VEL
LIN {X 0,Y 495.476,Z 899.154,A -85,B 0,C 180,E1 22974.132,E2 22974.132} C_VEL
LIN {X 0,Y 494.911,Z 918.15,A -85,B 0,C 180,E1 22973.641,E2 22973.641} C_VEL
LIN {X 0,Y 494.226,Z 936.46,A -85,B 0,C 180,E1 22972.952,E2 22972.952} C_VEL
LIN {X 0,Y 493.437,Z 954.205,A -85,B 0,C 180,E1 22972.064,E2 22972.064} C_VEL
LIN {X 0,Y 492.507,Z 971.704,A -85,B 0,C 180,E1 22970.955,E2 22970.955} C_VEL
LIN {X 0,Y 491.63,Z 988.064,A -85,B 0,C 180,E1 22969.673,E2 22969.673} C_VEL
LIN {X 0,Y 490.742,Z 1003.897,A -85,B 0,C 180,E1 22968.164,E2 22968.164} C_VEL
LIN {X 0,Y 489.981,Z 1017.544,A -85,B 0,C 180,E1 22966.6,E2 22966.6} C_VEL
LIN {X 0,Y 489.303,Z 1030.656,A -85,B 0,C 180,E1 22964.799,E2 22964.799} C_VEL
LIN {X 0,Y 488.764,Z 1042.174,A -85,B 0,C 180,E1 22962.884,E2 22962.884} C_VEL
LIN {X 0,Y 488.388,Z 1051.567,A -85,B 0,C 180,E1 22960.976,E2 22960.976} C_VEL
LIN {X 0,Y 488.145,Z 1059.085,A -85,B 0,C 180,E1 22959.075,E2 22959.075} C_VEL
LIN {X 0,Y 488.004,Z 1065.107,A -85,B 0,C 180,E1 22957.062,E2 22957.062} C_VEL
LIN {X 0,Y 487.931,Z 1069.668,A -85,B 0,C 180,E1 22954.938,E2 22954.938} C_VEL
LIN {X 0,Y 487.911,Z 1072.678,A -85,B 0,C 180,E1 22952.702,E2 22952.702} C_VEL
LIN {X 0,Y 487.909,Z 1073.916,A -85,B 0,C 180,E1 22950.47,E2 22950.47} C_VEL
LIN {X 0,Y 487.912,Z 1073.412,A -85,B 0,C 180,E1 22948.239,E2 22948.239} C_VEL
LIN {X 0,Y 487.924,Z 1071.158,A -85,B 0,C 180,E1 22946.005,E2 22946.005} C_VEL
LIN {X 0,Y 487.964,Z 1067.35,A -85,B 0,C 180,E1 22943.884,E2 22943.884} C_VEL
LIN {X 0,Y 488.073,Z 1061.799,A -85,B 0,C 180,E1 22941.755,E2 22941.755} C_VEL
LIN {X 0,Y 488.267,Z 1055.084,A -85,B 0,C 180,E1 22939.857,E2 22939.857} C_VEL
LIN {X 0,Y 488.602,Z 1045.893,A -85,B 0,C 180,E1 22937.832,E2 22937.832} C_VEL
LIN {X 0,Y 489.083,Z 1035.195,A -85,B 0,C 180,E1 22935.92,E2 22935.92} C_VEL
LIN {X 0,Y 489.692,Z 1022.785,A -85,B 0,C 180,E1 22934.09,E2 22934.09} C_VEL
LIN {X 0,Y 490.427,Z 1009.323,A -85,B 0,C 180,E1 22932.438,E2 22932.438} C_VEL
LIN {X 0,Y 491.239,Z 994.632,A -85,B 0,C 180,E1 22930.933,E2 22930.933} C_VEL
LIN {X 0,Y 492.086,Z 979.085,A -85,B 0,C 180,E1 22929.609,E2 22929.609} C_VEL
LIN {X 0,Y 492.953,Z 962.698,A -85,B 0,C 180,E1 22928.462,E2 22928.462} C_VEL
LIN {X 0,Y 493.791,Z 945.634,A -85,B 0,C 180,E1 22927.499,E2 22927.499} C_VEL
LIN {X 0,Y 494.508,Z 927.828,A -85,B 0,C 180,E1 22926.716,E2 22926.716} C_VEL
LIN {X 0,Y 495.147,Z 909.2,A -85,B 0,C 180,E1 22926.121,E2 22926.121} C_VEL
LIN {X 0,Y 495.571,Z 889.953,A -85,B 0,C 180,E1 22925.726,E2 22925.726} C_VEL
LIN {X 0,Y 496.951,Z 706.154,A -85,B 0,C 180,E1 22923.03,E2 22923.03} C_VEL
LIN {X 0,Y 495.075,Z 692.121,A -85,B 0,C 180,E1 22922.701,E2 22922.701} C_VEL
LIN {X 0,Y 497.023,Z 648.864,A -85,B 0,C 180,E1 22919.204,E2 22919.204} C_VEL
LIN {X 0,Y 498.38,Z 622.506,A -85,B 0,C 180,E1 22916.992,E2 22916.992} C_VEL
LIN {X 0,Y 491.646,Z 603.081,A -85,B 0,C 180,E1 22914.72,E2 22914.72} C_VEL
LIN {X 0,Y 488.812,Z 595.117,A -85,B 0,C 180,E1 22913.677,E2 22913.677} C_VEL
LIN {X 0,Y 488.839,Z 594.904,A -85,B 0,C 180,E1 22910.345,E2 22910.345} C_VEL
LIN {X 0,Y 488.775,Z 594.91,A -85,B 0,C 180,E1 22906.902,E2 22906.902} C_VEL
LIN {X 0,Y 488.795,Z 594.913,A -85,B 0,C 180,E1 22903.417,E2 22903.417} C_VEL
LIN {X 0,Y 488.839,Z 594.907,A -85,B 0,C 180,E1 22899.913,E2 22899.913} C_VEL
LIN {X 0,Y 488.777,Z 594.91,A -85,B 0,C 180,E1 22896.492,E2 22896.492} C_VEL
LIN {X 0,Y 488.791,Z 594.909,A -85,B 0,C 180,E1 22892.965,E2 22892.965} C_VEL
LIN {X 0,Y 488.838,Z 594.906,A -85,B 0,C 180,E1 22889.534,E2 22889.534} C_VEL
LIN {X 0,Y 488.782,Z 594.909,A -85,B 0,C 180,E1 22886.091,E2 22886.091} C_VEL
LIN {X 0,Y 488.784,Z 594.911,A -85,B 0,C 180,E1 22882.49,E2 22882.49} C_VEL
LIN {X 0,Y 488.831,Z 594.898,A -85,B 0,C 180,E1 22879.095,E2 22879.095} C_VEL
LIN {X 0,Y 488.784,Z 594.906,A -85,B 0,C 180,E1 22875.665,E2 22875.665} C_VEL
LIN {X 0,Y 488.788,Z 594.911,A -85,B 0,C 180,E1 22872.043,E2 22872.043} C_VEL
LIN {X 0,Y 488.833,Z 594.896,A -85,B 0,C 180,E1 22868.587,E2 22868.587} C_VEL
LIN {X 0,Y 488.79,Z 594.9,A -85,B 0,C 180,E1 22865.164,E2 22865.164} C_VEL
LIN {X 0,Y 488.788,Z 594.908,A -85,B 0,C 180,E1 22861.524,E2 22861.524} C_VEL
LIN {X 0,Y 488.831,Z 594.904,A -85,B 0,C 180,E1 22858.124,E2 22858.124} C_VEL
LIN {X 0,Y 488.802,Z 594.898,A -85,B 0,C 180,E1 22854.601,E2 22854.601} C_VEL
LIN {X 0,Y 488.791,Z 594.899,A -85,B 0,C 180,E1 22851.056,E2 22851.056} C_VEL
LIN {X 0,Y 488.832,Z 594.905,A -85,B 0,C 180,E1 22847.598,E2 22847.598} C_VEL
LIN {X 0,Y 488.817,Z 594.906,A -85,B 0,C 180,E1 22844.023,E2 22844.023} C_VEL
LIN {X 0,Y 488.795,Z 594.908,A -85,B 0,C 180,E1 22840.523,E2 22840.523} C_VEL
LIN {X 0,Y 488.828,Z 594.906,A -85,B 0,C 180,E1 22836.991,E2 22836.991} C_VEL
LIN {X 0,Y 488.831,Z 594.904,A -85,B 0,C 180,E1 22833.36,E2 22833.36} C_VEL
LIN {X 0,Y 488.799,Z 594.909,A -85,B 0,C 180,E1 22829.913,E2 22829.913} C_VEL
LIN {X 0,Y 488.819,Z 594.906,A -85,B 0,C 180,E1 22826.336,E2 22826.336} C_VEL
LIN {X 0,Y 488.83,Z 594.906,A -85,B 0,C 180,E1 22822.718,E2 22822.718} C_VEL
LIN {X 0,Y 488.86,Z 595.239,A -85,B 0,C 180,E1 22822.034,E2 22822.034} C_VEL
LIN {X 0,Y 493.593,Z 611.466,A -85,B 0,C 180,E1 22819.363,E2 22819.363} C_VEL
LIN {X 0,Y 495.012,Z 618.067,A -85,B 0,C 180,E1 22818.353,E2 22818.353} C_VEL
LIN {X 0,Y 493.388,Z 646.84,A -85,B 0,C 180,E1 22814.603,E2 22814.603} C_VEL
LIN {X 0,Y 491.95,Z 676.647,A -85,B 0,C 180,E1 22810.801,E2 22810.801} C_VEL
LIN {X 0,Y 491.131,Z 696.112,A -85,B 0,C 180,E1 22808.346,E2 22808.346} C_VEL
LIN {X 0,Y 490.018,Z 699.924,A -85,B 0,C 180,E1 22807.915,E2 22807.915} C_VEL
LIN {X 0,Y 486.134,Z 706.893,A -85,B 0,C 180,E1 22807.338,E2 22807.338} C_VEL
LIN {X 0,Y 484.296,Z 712.181,A -85,B 0,C 180,E1 22807.061,E2 22807.061} C_VEL
LIN {X 0,Y 484.283,Z 715.766,A -85,B 0,C 180,E1 22806.942,E2 22806.942} C_VEL
LIN {X 0,Y 485.463,Z 724.566,A -85,B 0,C 180,E1 22806.744,E2 22806.744} C_VEL
LIN {X 0,Y 484.385,Z 825.334,A -85,B 0,C 180,E1 22805.141,E2 22805.141} C_VEL
LIN {X 0,Y 484.085,Z 840.825,A -85,B 0,C 180,E1 22804.663,E2 22804.663} C_VEL
LIN {X 0,Y 483.597,Z 856.084,A -85,B 0,C 180,E1 22803.934,E2 22803.934} C_VEL
LIN {X 0,Y 483.027,Z 869.674,A -85,B 0,C 180,E1 22803.034,E2 22803.034} C_VEL
LIN {X 0,Y 482.445,Z 881.959,A -85,B 0,C 180,E1 22801.973,E2 22801.973} C_VEL
LIN {X 0,Y 481.885,Z 893.485,A -85,B 0,C 180,E1 22800.692,E2 22800.692} C_VEL
LIN {X 0,Y 481.343,Z 903.55,A -85,B 0,C 180,E1 22799.256,E2 22799.256} C_VEL
LIN {X 0,Y 480.923,Z 911.758,A -85,B 0,C 180,E1 22797.756,E2 22797.756} C_VEL
LIN {X 0,Y 480.607,Z 918.956,A -85,B 0,C 180,E1 22796.007,E2 22796.007} C_VEL
LIN {X 0,Y 480.413,Z 924.139,A -85,B 0,C 180,E1 22794.205,E2 22794.205} C_VEL
LIN {X 0,Y 480.319,Z 927.328,A -85,B 0,C 180,E1 22792.443,E2 22792.443} C_VEL
LIN {X 0,Y 480.282,Z 928.853,A -85,B 0,C 180,E1 22790.599,E2 22790.599} C_VEL
LIN {X 0,Y 480.282,Z 928.492,A -85,B 0,C 180,E1 22788.696,E2 22788.696} C_VEL
LIN {X 0,Y 480.322,Z 926.439,A -85,B 0,C 180,E1 22786.943,E2 22786.943} C_VEL
LIN {X 0,Y 480.427,Z 922.712,A -85,B 0,C 180,E1 22785.202,E2 22785.202} C_VEL
LIN {X 0,Y 480.624,Z 917.099,A -85,B 0,C 180,E1 22783.473,E2 22783.473} C_VEL
LIN {X 0,Y 480.928,Z 910.033,A -85,B 0,C 180,E1 22781.878,E2 22781.878} C_VEL
LIN {X 0,Y 481.351,Z 901.584,A -85,B 0,C 180,E1 22780.411,E2 22780.411} C_VEL
LIN {X 0,Y 481.85,Z 891.742,A -85,B 0,C 180,E1 22779.073,E2 22779.073} C_VEL
LIN {X 0,Y 482.374,Z 880.529,A -85,B 0,C 180,E1 22777.863,E2 22777.863} C_VEL
LIN {X 0,Y 482.982,Z 867.498,A -85,B 0,C 180,E1 22776.777,E2 22776.777} C_VEL
LIN {X 0,Y 483.501,Z 854.223,A -85,B 0,C 180,E1 22775.935,E2 22775.935} C_VEL
LIN {X 0,Y 483.948,Z 839.585,A -85,B 0,C 180,E1 22775.258,E2 22775.258} C_VEL
LIN {X 0,Y 484.252,Z 823.483,A -85,B 0,C 180,E1 22774.782,E2 22774.782} C_VEL
LIN {X 0,Y 485.016,Z 721.325,A -85,B 0,C 180,E1 22773.183,E2 22773.183} C_VEL
LIN {X 0,Y 482.86,Z 708.743,A -85,B 0,C 180,E1 22772.848,E2 22772.848} C_VEL
LIN {X 0,Y 484.035,Z 679.531,A -85,B 0,C 180,E1 22769.171,E2 22769.171} C_VEL
LIN {X 0,Y 485.453,Z 650.67,A -85,B 0,C 180,E1 22765.468,E2 22765.468} C_VEL
LIN {X 0,Y 487.067,Z 621.585,A -85,B 0,C 180,E1 22761.675,E2 22761.675} C_VEL
LIN {X 0,Y 487.111,Z 618.521,A -85,B 0,C 180,E1 22761.263,E2 22761.263} C_VEL
LIN {X 0,Y 482.097,Z 600.253,A -85,B 0,C 180,E1 22758.394,E2 22758.394} C_VEL
LIN {X 0,Y 480.893,Z 595.974,A -85,B 0,C 180,E1 22757.634,E2 22757.634} C_VEL
LIN {X 0,Y 480.879,Z 595.894,A -85,B 0,C 180,E1 22754.07,E2 22754.07} C_VEL
LIN {X 0,Y 480.887,Z 595.891,A -85,B 0,C 180,E1 22750.442,E2 22750.442} C_VEL
LIN {X 0,Y 480.886,Z 595.871,A -85,B 0,C 180,E1 22746.782,E2 22746.782} C_VEL
LIN {X 0,Y 480.877,Z 595.897,A -85,B 0,C 180,E1 22743.126,E2 22743.126} C_VEL
LIN {X 0,Y 480.874,Z 595.866,A -85,B 0,C 180,E1 22739.513,E2 22739.513} C_VEL
LIN {X 0,Y 480.888,Z 595.894,A -85,B 0,C 180,E1 22735.992,E2 22735.992} C_VEL
LIN {X 0,Y 480.888,Z 595.889,A -85,B 0,C 180,E1 22732.317,E2 22732.317} C_VEL
LIN {X 0,Y 480.867,Z 595.897,A -85,B 0,C 180,E1 22728.766,E2 22728.766} C_VEL
LIN {X 0,Y 480.883,Z 595.891,A -85,B 0,C 180,E1 22725.155,E2 22725.155} C_VEL
LIN {X 0,Y 480.888,Z 595.88,A -85,B 0,C 180,E1 22721.538,E2 22721.538} C_VEL
LIN {X 0,Y 480.872,Z 595.897,A -85,B 0,C 180,E1 22717.986,E2 22717.986} C_VEL
LIN {X 0,Y 480.862,Z 595.884,A -85,B 0,C 180,E1 22714.362,E2 22714.362} C_VEL
LIN {X 0,Y 480.896,Z 595.891,A -85,B 0,C 180,E1 22710.762,E2 22710.762} C_VEL
LIN {X 0,Y 480.891,Z 595.88,A -85,B 0,C 180,E1 22707.087,E2 22707.087} C_VEL
LIN {X 0,Y 480.859,Z 595.892,A -85,B 0,C 180,E1 22703.51,E2 22703.51} C_VEL
LIN {X 0,Y 480.867,Z 595.89,A -85,B 0,C 180,E1 22699.938,E2 22699.938} C_VEL
LIN {X 0,Y 480.893,Z 595.884,A -85,B 0,C 180,E1 22696.302,E2 22696.302} C_VEL
LIN {X 0,Y 480.879,Z 595.9,A -85,B 0,C 180,E1 22692.733,E2 22692.733} C_VEL
LIN {X 0,Y 480.85,Z 595.88,A -85,B 0,C 180,E1 22689.214,E2 22689.214} C_VEL
LIN {X 0,Y 480.886,Z 595.891,A -85,B 0,C 180,E1 22685.728,E2 22685.728} C_VEL
LIN {X 0,Y 480.887,Z 595.884,A -85,B 0,C 180,E1 22682.145,E2 22682.145} C_VEL
LIN {X 0,Y 480.845,Z 595.889,A -85,B 0,C 180,E1 22678.69,E2 22678.69} C_VEL
LIN {X 0,Y 480.87,Z 595.891,A -85,B 0,C 180,E1 22675.11,E2 22675.11} C_VEL
LIN {X 0,Y 480.896,Z 595.884,A -85,B 0,C 180,E1 22671.632,E2 22671.632} C_VEL
LIN {X 0,Y 480.847,Z 595.9,A -85,B 0,C 180,E1 22668.12,E2 22668.12} C_VEL
LIN {X 0,Y 480.857,Z 595.888,A -85,B 0,C 180,E1 22664.565,E2 22664.565} C_VEL
LIN {X 0,Y 480.896,Z 595.89,A -85,B 0,C 180,E1 22661.074,E2 22661.074} C_VEL
LIN {X 0,Y 480.844,Z 595.895,A -85,B 0,C 180,E1 22657.634,E2 22657.634} C_VEL
LIN {X 0,Y 480.844,Z 595.888,A -85,B 0,C 180,E1 22653.976,E2 22653.976} C_VEL
LIN {X 0,Y 480.9,Z 595.89,A -85,B 0,C 180,E1 22650.478,E2 22650.478} C_VEL
LIN {X 0,Y 480.869,Z 595.9,A -85,B 0,C 180,E1 22646.925,E2 22646.925} C_VEL
LIN {X 0,Y 480.837,Z 595.9,A -85,B 0,C 180,E1 22643.385,E2 22643.385} C_VEL
